// TwinCAT 3 PLC project protobuf
// Title: protobuf
// Company: TcHaxx
// Author: densogiaichned
// ProjectVersion: 0.0.1.0
// Description: Protocol Buffers for TwinCAT 3
// ProgramVersion: 3.1.4026.23
// libraries:
//   snappy, * (TcHaxx)
//   Tc2_Standard, * (Beckhoff Automation GmbH)
//   Tc2_System, * (Beckhoff Automation GmbH)
//   Tc2_Utilities, * (Beckhoff Automation GmbH)
//   TcUnit, * (www.tcunit.org)
// project tree:
//   DUTs/ E_CodedInputStreamErrorCode.TcDUT, E_CodedOutputStreamErrorCode.TcDUT, ST_ParseContext.TcDUT, ST_WriteContext.TcDUT, ST_Span.TcDUT, T_ProtobufMaxString.TcDUT, T_ProtobufRawBuffer.TcDUT
//   FieldCodec/ FB_FieldCodec.TcPOU, FB_FieldCodecFixed32.TcPOU, FB_FieldCodecFixed64.TcPOU, FB_FieldCodecDouble.TcPOU, FB_FieldCodecBool.TcPOU, FB_FieldCodecEnum.TcPOU, FB_FieldCodecMessage.TcPOU, FB_FieldCodecUInt64.TcPOU, FB_FieldCodecUInt32.TcPOU, FB_FieldCodecString.TcPOU, FB_FieldCodecFloat.TcPOU, FB_FieldCodecInt32.TcPOU, FB_FieldCodecSint32.TcPOU, FB_FieldCodecInt64.TcPOU, FB_FieldCodecSint64.TcPOU, FB_FieldCodecBytes.TcPOU
//   GVLs/ GCL_PB.TcGVL, Param_PB.TcGVL
//   Helper/DUTs/ ST_VariableLengthArrayInfo.TcDUT, T_AnyInt.TcDUT, T_AnyIntOrBit.TcDUT, T_AnyString.TcDUT, T_AnyNum.TcDUT, T_Any.TcDUT, T_AnyBit.TcDUT, T_AnyBytes.TcDUT
//   Helper/POUs/ F_ParseError.TcPOU, F_WriteError.TcPOU, F_ToAnyBit.TcPOU, F_ToAnyInt.TcPOU, F_ToAnyBytes.TcPOU, F_ToAnyType.TcPOU, F_ToAnyNum.TcPOU, F_ToAnyString.TcPOU, F_BufferInfo.TcPOU, F_WriteToBuffer.TcPOU, F_ReadFromBuffer.TcPOU
//   ITFs/ I_Message.TcIO, I_FieldCodec.TcIO, I_RepeatedField.TcIO, I_ValueReader.TcIO, I_ValueWriter.TcIO
//   ParsingPrimitivesMessages/POUs/ F_ReadMessage.TcPOU, F_ReadRawMessage.TcPOU, F_SkipLastField.TcPOU, F_CheckReadEndOfStreamTag.TcPOU
//   ParsingPrimitives/DUTs/ E_ParserErrorCode.TcDUT, ST_ParserInternalState.TcDUT
//   ParsingPrimitives/POUs/ F_DecodeZigZag32.TcPOU, F_DecodeZigZag64.TcPOU, F_MaybeConsumeTag.TcPOU, F_ParseDouble.TcPOU, F_ParseFloat.TcPOU, F_ParseRawLittleEndian32.TcPOU, F_ParseLength.TcPOU, F_ParseRawLittleEndian64.TcPOU, F_ParseRawVarint64.TcPOU, F_ParseTag.TcPOU, F_ParseRawVarint32.TcPOU, F_PeekTag.TcPOU, F_ReadBytes.TcPOU, F_ReadRawByte.TcPOU, F_ReadRawBytes.TcPOU, F_ReadStringInternal.TcPOU, F_SkipRawBytes.TcPOU, F_ReadRawString.TcPOU, F_ReadString.TcPOU
//   / PlcTask.TcTTO, PlcTaskUnitTests.TcTTO
//   POUs/ComputeSize/ F_ComputeBoolSize.TcPOU, F_ComputeMessageSize.TcPOU, F_ComputeTagSize.TcPOU, F_ComputeStringSize.TcPOU, F_ComputeFixed32Size.TcPOU, F_ComputeSFixed32Size.TcPOU, F_ComputeFixed64Size.TcPOU, F_ComputeSFixed64Size.TcPOU, F_ComputeInt32Size.TcPOU, F_ComputeEnumSize.TcPOU, F_ComputeFloatSize.TcPOU, F_ComputeDoubleSize.TcPOU, F_ComputeInt64Size.TcPOU, F_ComputeLengthSize.TcPOU, F_ComputeBytesSize.TcPOU, F_ComputeRawVarint64Size.TcPOU, F_ComputeSInt64Size.TcPOU, F_ComputeUInt32Size.TcPOU, F_ComputeRawVarint32Size.TcPOU, F_ComputeSInt32Size.TcPOU, F_ComputeUInt64Size.TcPOU
//   POUs/ FB_MessageParser.TcPOU, FB_MessageWriter.TcPOU
//   POUs/ParseContext/ FB_ParseContext.TcPOU
//   POUs/SegmentedBufferHelper/ F_SbhIsReachedLimit.TcPOU, F_SbhPushLimit.TcPOU, F_SbhPopLimit.TcPOU, F_SbhRecomputeBufferSizeAfterLimit.TcPOU
//   POUs/Span/ F_SpanFromArray.TcPOU, F_SpanSlice.TcPOU
//   POUs/WriteContext/ FB_WriteContext.TcPOU
//   Project Information/ F_GetCompany.TcPOU, F_GetTitle.TcPOU, F_GetVersion.TcPOU
//   RepeatedField/ FB_RepeatedField.TcPOU, F_IsPackedRepeatedField.TcPOU, F_ReadRepeatedField.TcPOU, F_WriteRepeatedField.TcPOU
//   WireFormat/DUTs/ E_WireType.TcDUT
//   WireFormat/GCLs/ GCL_WireFormat.TcGVL
//   WireFormat/POus/ F_GetTagFieldNumber.TcPOU, F_GetTagWireType.TcPOU, F_MakeTag.TcPOU
//   WritingPrimitivesMessages/POUs/ F_SetMessageValue.TcPOU, F_WriteMessage.TcPOU, F_WriteRawMessage.TcPOU
//   WritingPrimitives/DUTs/ E_WriterErrorCode.TcDUT, ST_WriterInternalState.TcDUT
//   WritingPrimitives/POUs/ F_EncodeZigZag32.TcPOU (not stored), F_EncodeZigZag64.TcPOU (not stored), F_WriteBytes.TcPOU, F_WriteDouble.TcPOU, F_WriteFixed32.TcPOU (not stored), F_WriteRawByte.TcPOU, F_WriteSInt32.TcPOU, F_WriteSFixed32.TcPOU (not stored), F_WriteFloat.TcPOU (not stored), F_WriteInt32.TcPOU, F_WriteFixed64.TcPOU (not stored), F_WriteSFixed64.TcPOU (not stored), F_WriteSInt64.TcPOU, F_WriteRawString.TcPOU (not stored), F_WriteRawTag.TcPOU (not stored), F_WriteUInt32.TcPOU (not stored), F_WriteRawLittleEndian32.TcPOU, F_WriteLength.TcPOU, F_WriteRawBytes.TcPOU, F_WriteRawLittleEndian64.TcPOU, F_WriteRawVarint32.TcPOU, F_WriteRawVarint64.TcPOU (not stored), F_WriteString.TcPOU (not stored), F_WriteTag.TcPOU (not stored), F_WriteEnum.TcPOU, F_WriteUInt64.TcPOU (not stored), F_WriteInt64.TcPOU
//   __TESTs/EnumTests/DUTs/ E_INT.TcDUT, E_BYTE.TcDUT
//   __TESTs/EnumTests/ FB_F_ComputeEnumSizeTests.TcPOU, FB_ReadEnumTests.TcPOU, FB_WriteEnumTests.TcPOU, PRG_EnumTests.TcPOU
//   __TESTs/HelperTests/ FB_F_ToAnyBytesTests.TcPOU, PRG_HelperTests.TcPOU
//   __TESTs/MessagesTests/Complex/ FB_ComplexDataTests.TcPOU, FB_RepeatedComplexDataTests.TcPOU, FB_DeviceTests.TcPOU, FB_MotorTests.TcPOU
//   __TESTs/MessagesTests/Complex/_gen/ E_Color.TcDUT, E_DataType.TcDUT, E_Status.TcDUT, FB_ComplexData.TcPOU, FB_Device.TcPOU, FB_Motor.TcPOU, FB_MotorConfig.TcPOU, FB_RepeatedComplexData.TcPOU, FB_SensorReading.TcPOU, ST_ComplexData.TcDUT, ST_Device.TcDUT, ST_Motor.TcDUT, ST_MotorConfig.TcDUT, ST_RepeatedComplexData.TcDUT, ST_SensorReading.TcDUT
//   __TESTs/MessagesTests/DUTs/ ST_Example.TcDUT
//   __TESTs/MessagesTests/FooBarBaz/ FB_FooBarBazTests.TcPOU
//   __TESTs/MessagesTests/FooBarBaz/_gen/ FB_Bar.TcPOU, FB_Baz.TcPOU, FB_Foo.TcPOU, ST_Bar.TcDUT, ST_Baz.TcDUT, ST_Foo.TcDUT
//   __TESTs/MessagesTests/POUs/ FB_ExampleMessage.TcPOU, FB_RoundTripMessageExampleTest.TcPOU
//   __TESTs/MessagesTests/ PRG_MessageTests.TcPOU
//   __TESTs/MessagesTests/Scalars/ FB_ScalarTypesTest.TcPOU
//   __TESTs/MessagesTests/Scalars/_gen/ FB_ScalarTypes.TcPOU, ST_ScalarTypes.TcDUT
//   __TESTs/ParsingPrimitivesTests/ FB_DecodeZigZag32Tests.TcPOU (not stored), FB_DecodeZigZag64Tests.TcPOU (not stored), FB_ParseDoubleTests.TcPOU, FB_ParseFloatTests.TcPOU, FB_ParseRawVarint32Tests.TcPOU, FB_ParseRawVarint64Tests.TcPOU, FB_ReadBytesTests.TcPOU, FB_ReadRawStringTests.TcPOU, FB_ReadStringTests.TcPOU, PRG_ParsingPrimitiveTests.TcPOU
//   __TESTs/ PRG_UnitTests.TcPOU
//   Version/ Global_Version.TcGVL
//   __TESTs/RepeatedFieldTests/ PRG_RepeatedFieldTests.TcPOU
//   __TESTs/RepeatedFieldTests/Read/ FB_ReadRepeatedFieldEnumTests.TcPOU, FB_ReadRepeatedFieldBoolTests.TcPOU, FB_ReadRepeatedFieldBytesTests.TcPOU, FB_ReadRepeatedFieldFixed32Tests.TcPOU, FB_ReadRepeatedFieldFixed64Tests.TcPOU, FB_ReadRepeatedFieldStringTests.TcPOU, FB_ReadRepeatedFieldUint32Tests.TcPOU, PRG_ReadRepeatedFieldTests.TcPOU
//   __TESTs/RepeatedFieldTests/RoundTrip/ FB_RoundTripRepeatedFieldUInt32Tests.TcPOU, FB_RoundTripRepeatedFieldStringTests.TcPOU, FB_RoundTripRepeatedFieldUInt64Tests.TcPOU, PRG_RoundTripRepeatedFieldTests.TcPOU
//   __TESTs/RepeatedFieldTests/Write/ FB_WriteRepeatedFieldBoolTests.TcPOU, FB_WriteRepeatedFieldBytesTests.TcPOU, FB_WriteRepeatedFieldDoubleTests.TcPOU, FB_WriteRepeatedFieldFixed32Tests.TcPOU, FB_WriteRepeatedFieldFixed64Tests.TcPOU, FB_WriteRepeatedFieldFloatTests.TcPOU, FB_WriteRepeatedFieldInt32Tests.TcPOU, FB_WriteRepeatedFieldInt64Tests.TcPOU, FB_WriteRepeatedFieldMessageTests.TcPOU, FB_WriteRepeatedFieldSInt32Tests.TcPOU, FB_WriteRepeatedFieldSInt64Tests.TcPOU, FB_WriteRepeatedFieldStringTests.TcPOU, FB_WriteRepeatedFieldUint32Tests.TcPOU, FB_WriteRepeatedFieldUint64Tests.TcPOU, PRG_WriteRepeatedFieldTests.TcPOU
//   __TESTs/RoundTripTests/ FB_RoundTripBytesTests.TcPOU, FB_RoundTripFloatTests.TcPOU, FB_RoundTripDoubleTests.TcPOU, FB_RoundTripRawVarint32Tests.TcPOU, FB_RoundTripRawVarint64Tests.TcPOU, FB_RoundTripStringTests.TcPOU, FB_RoundTripTagTests.TcPOU, FB_RoundTripZigZag32Tests.TcPOU, FB_RoundTripZigZag64Tests.TcPOU, PRG_RoundTripTests.TcPOU
//   __TESTs/SpanTests/ FB_F_SpanFromArrayTests.TcPOU, FB_F_SpanSliceTests.TcPOU, PRG_SpanTests.TcPOU
//   __TESTs/WireFormatTests/ FB_MakeTagTests.TcPOU, PRG_WireFormatTests.TcPOU
//   __TESTs/WritingPrimitiveTests/ FB_EncodeZigZag64Tests.TcPOU (not stored), FB_EncodeZigZag32Tests.TcPOU, FB_WriteBytesTests.TcPOU, FB_WriteDoubleTests.TcPOU, FB_WriteRawVarint32Tests.TcPOU, FB_WriteFloatTests.TcPOU, FB_WriteRawVarint64Tests.TcPOU, FB_WriteTagTests.TcPOU, FB_WriteStringTests.TcPOU, PRG_WritingPrimitiveTests.TcPOU
//   __TESTs/_ISSUES/ FB_Issue4Tests.TcPOU, PRG_IssuesTests.TcPOU
//   __TESTs/_ISSUES/_gen/ E_EnumOfTypeSint.TcDUT, FB_RepeatedEnumTests.TcPOU, ST_RepeatedEnumTests.TcDUT
// real-time tasks:
//   TASK PlcTask: cycle T#10ms, priority 8, ADS port 350
//   TASK PlcTaskUnitTests: cycle T#10ms, priority 6, ADS port 351

CONFIGURATION protobuf
    RESOURCE PLC ON TwinCAT3
        TASK PlcTask(INTERVAL := T#10ms, PRIORITY := 8);
        TASK PlcTaskUnitTests(INTERVAL := T#10ms, PRIORITY := 6);
        PROGRAM PRG_UnitTests WITH PlcTaskUnitTests : PRG_UnitTests;
    END_RESOURCE
END_CONFIGURATION

// ---- DUTs/E_CodedInputStreamErrorCode.TcDUT
{attribute 'qualified_only'}
{attribute 'strict'}
{attribute 'to_string'}
TYPE E_CodedInputStreamErrorCode :
(
	NoError := S_OK,            // No Error.
    BUFFER_LOWER_BOUND := -1,   // Invalid lower bound for buffer.
    BUFFER_SIZE := -2           // Invalid size of buffer (0 >= size > Param.cMaxProtobufRawBuffer).
) DINT;
END_TYPE

// ---- DUTs/E_CodedOutputStreamErrorCode.TcDUT
{attribute 'qualified_only'}
{attribute 'strict'}
{attribute 'to_string'}
TYPE E_CodedOutputStreamErrorCode :
(
	NoError := S_OK,            // No Error.
    BUFFER_LOWER_BOUND := -1,   // Invalid lower bound for buffer.
    BUFFER_SIZE := -2           // Invalid size of buffer (0 >= size > Param.cMaxProtobufRawBuffer).
) DINT;
END_TYPE

// ---- DUTs/ST_ParseContext.TcDUT
TYPE ST_ParseContext :
STRUCT
    stBuffer    	: ST_Span;
    stState     	: ST_ParserInternalState;
	pCurrentContext : POINTER TO FB_ParseContext; 	// The current context we are operating on
END_STRUCT
END_TYPE

// ---- DUTs/ST_WriteContext.TcDUT
// An opaque struct that represents the current serialization state and is passed along as the serialization proceeds.
TYPE ST_WriteContext :
STRUCT
    stBuffer    	: ST_Span;
    stState     	: ST_WriterInternalState;
	pCurrentContext : POINTER TO FB_WriteContext;	// The current context we are operating on
END_STRUCT
END_TYPE

// ---- DUTs/ST_Span.TcDUT
TYPE ST_Span :
STRUCT
    pBuffer     : POINTER TO BYTE;
    nSize       : UDINT;
END_STRUCT
END_TYPE

// ---- DUTs/T_ProtobufMaxString.TcDUT
TYPE T_ProtobufMaxString : STRING(Param_PB.cMaxCharacter + 1); END_TYPE

// ---- DUTs/T_ProtobufRawBuffer.TcDUT
TYPE T_ProtobufRawBuffer : ARRAY[0..Param_PB.cMaxProtobufRawBuffer] OF BYTE; END_TYPE

// ---- Helper/DUTs/ST_VariableLengthArrayInfo.TcDUT
TYPE ST_VariableLengthArrayInfo :
STRUCT
    nLowerBound : DINT;
    nUpperBound : DINT;
    nSize       : UDINT;
END_STRUCT
END_TYPE

// ---- Helper/DUTs/T_AnyInt.TcDUT
TYPE T_AnyInt : __SYSTEM.AnyType; END_TYPE

// ---- Helper/DUTs/T_AnyIntOrBit.TcDUT
TYPE T_AnyIntOrBit : __SYSTEM.AnyType; END_TYPE

// ---- Helper/DUTs/T_AnyString.TcDUT
TYPE T_AnyString : __SYSTEM.AnyType; END_TYPE

// ---- Helper/DUTs/T_AnyNum.TcDUT
TYPE T_AnyNum : __SYSTEM.AnyType; END_TYPE

// ---- Helper/DUTs/T_Any.TcDUT
TYPE T_Any : __SYSTEM.AnyType; END_TYPE

// ---- Helper/DUTs/T_AnyBit.TcDUT
TYPE T_AnyBit : __SYSTEM.AnyType; END_TYPE

// ---- Helper/DUTs/T_AnyBytes.TcDUT
TYPE T_AnyBytes : __SYSTEM.AnyType; END_TYPE

// ---- ParsingPrimitives/DUTs/E_ParserErrorCode.TcDUT
// Parser ErrorCode is set when a message being parsed is invalid in some way,
// e.g. malformed Varint. Zero means no error.
{attribute 'qualified_only'}
{attribute 'strict'}
{attribute 'to_string'}
TYPE E_ParserErrorCode :
(
	NoError := S_OK,                // No Error.
    InternalError := -1,            // Internal parser error.
    MalformedVarInt := -2,          // Encountered a malformed Varint.
    InvalidDataType := -3,          // Datatype not supported, e.g. F_ParseRawInt32 -> LINT
    TruncatedMessage := -4,         // While parsing a protocol message, the input ended unexpectedly in the middle of a field.  This could mean either that the input has been truncated or that an embedded message misreported its own length.
    InvalidUtf8 := -5,              //
    NotEnoughMem := -6,             // e.g. Array [0..15] OF BYTES but F_ReadRawBytes length is 32.
    EndOfStream := -7,              //
    MoreDataAvailable := -8,        // Completed reading a message while more data was available in the stream.
    RecursionLimitExceeded := -9,   // 
    NegativeSize := -10,            // Encountered an embedded string or message which claimed to have negative size.
    InvalidTag := -11,              // Protocol message contained an invalid tag (zero).
    InvalidWireType := -12,         // Protocol message contained a tag with an invalid wire type.
    NotImplemented := -999          // Not implemented yet.
) DINT := NoError;
END_TYPE

// ---- ParsingPrimitives/DUTs/ST_ParserInternalState.TcDUT
TYPE ST_ParserInternalState :
STRUCT
    nBufferSize             : UDINT;                        // Size of the current buffer
    nBufferPos              : UDINT;                        // The position within the current buffer (i.e. the next byte to read)
    nLastTag                : UDINT;                        // The last tag we read. 0 indicates we've read to the end of the stream (or haven't read anything yet).
    nNextTag                : UDINT;                        //
    nRecursionDepth         : UDINT;                        // Current recursion depth
    nRecursionLimit         : UDINT := Param_PB.cRecursionLimit; 
    nSizeLimit              : UDINT := Param_PB.cMaxProtobufRawBuffer;
    nBufferSizeAfterLimit   : UDINT;                        // If we are currently inside a length-delimited block, this is the number of bytes in the buffer that are still available once we leave the delimited block.
    nCurrentLimit           : UDINT := GCL_PB.cSbhLimit;    // The absolute position of the end of the current length-delimited block (including totalBytesRetired).
    nTotalBytesRetired      : UDINT;                        // The total number of consumed before the start of the current buffer.
    bError                  : BOOL;                         // True if error occured.
    bDiscardUnknownFields   : BOOL;                         // When set to true, unknown fields will be discarded while parsing.
    bHasNextTag             : BOOL; 
    eParserErrorCode        : E_ParserErrorCode;            // 0 = no error, <> 0 = error
END_STRUCT
END_TYPE

// ---- WireFormat/DUTs/E_WireType.TcDUT
// Wire types within protobuf encoding/decoding.
{attribute 'qualified_only'}
{attribute 'to_string'}
TYPE E_WireType :
(
	Varint := 0,            // Variable-length integer.
    Fixed64 := 1,           // Fixed-length 64-bit integer.
    LengthDelimited := 2,   // Length-delimited value, i.e. a length followed by that many bytes of data.
    StartGroup := 3,        // "start group" value
    EndGroup := 4,          // "end group" value
    Fixed32 := 5            // Fixed-length 32-bit value.
) UDINT;
END_TYPE

// ---- WritingPrimitives/DUTs/E_WriterErrorCode.TcDUT
// Wrtier ErrorCode is set when a message being written is invalid in some way,
// e.g. malformed Varint. Zero means no error.
{attribute 'qualified_only'}
{attribute 'strict'}
{attribute 'to_string'}
TYPE E_WriterErrorCode :
(
	NoError := S_OK,            // No Error.
    InternalError := -1,        // Internal writer error.
    MalformedVarInt := -2,      // Encountered a malformed Varint.
    InvalidDataType := -3,      // Datatype not supported, e.g. F_WriteVarInt32 -> LINT
    TruncatedMessage := -4,     // Not enough space left in given buffer
    InvalidUtf8 := -5,          //
    NotEnoughMem := -6          // e.g. Array [0..15] OF BYTES but F_ReadRawBytes length is 32.
) DINT := NoError;
END_TYPE

// ---- WritingPrimitives/DUTs/ST_WriterInternalState.TcDUT
TYPE ST_WriterInternalState :
STRUCT
    nBufferSize         : UDINT;                // Size of the current buffer
    nBufferPos          : UDINT;                // The position within the current buffer (i.e. the next byte to read)
    bError              : BOOL;
    eWriterErrorCode    : E_WriterErrorCode;    // 0 = no error, <> 0 = error
END_STRUCT
END_TYPE

// ---- __TESTs/EnumTests/DUTs/E_INT.TcDUT
{attribute 'qualified_only'}
{attribute 'strict'}
{attribute 'to_string'}
TYPE E_INT :
(	
	eMIN := -32768,
	eVAL0 := 0,
	eVAL1,
	eVAL2,
	eVAL3,
	eMAX := 32767
) INT;
END_TYPE

// ---- __TESTs/EnumTests/DUTs/E_BYTE.TcDUT
{attribute 'qualified_only'}
{attribute 'strict'}
{attribute 'to_string'}
TYPE E_BYTE :
(
	eMIN := 0,
	eVAL1,
	eVAL2,
	eVAL3,
	eMAX := 255
) BYTE;
END_TYPE

// ---- __TESTs/MessagesTests/Complex/_gen/E_Color.TcDUT
(*******************************************************************************
                          protoc-gen-twincat V0.0.0.0                           
                  https://github.com/TcHaxx/protoc-gen-twincat                  
*******************************************************************************)
{attribute 'qualified_only'}
{attribute 'strict'}
{attribute 'to_string'}
// Enum with enum_prefix and enum_integer_type options
TYPE E_Color :
(
	COLOR_DEFAULT := 0,
	COLOR_RED := 1,
	COLOR_GREEN := 2,
	COLOR_BLUE := 3
) WORD;
END_TYPE

// ---- __TESTs/MessagesTests/Complex/_gen/E_DataType.TcDUT
(*******************************************************************************
                          protoc-gen-twincat V0.0.0.0                           
                  https://github.com/TcHaxx/protoc-gen-twincat                  
*******************************************************************************)
{attribute 'qualified_only'}
{attribute 'strict'}
{attribute 'to_string'}
TYPE E_DataType :
(
	DATA_TYPE_UNKNOWN := 0,
	DATA_TYPE_TEMPERATURE := 1,
	DATA_TYPE_PRESSURE := 2,
	DATA_TYPE_HUMIDITY := 3
) BYTE;
END_TYPE

// ---- __TESTs/MessagesTests/Complex/_gen/E_Status.TcDUT
(*******************************************************************************
                          protoc-gen-twincat V0.0.0.0                           
                  https://github.com/TcHaxx/protoc-gen-twincat                  
*******************************************************************************)
{attribute 'qualified_only'}
{attribute 'strict'}
{attribute 'to_string'}
// Another enum for testing
TYPE E_Status :
(
	STATUS_IDLE := 0,
	STATUS_RUNNING := 1,
	STATUS_ERROR := 2
) DWORD;
END_TYPE

// ---- __TESTs/MessagesTests/Complex/_gen/ST_ComplexData.TcDUT
(*******************************************************************************
                          protoc-gen-twincat V0.0.0.0                           
                  https://github.com/TcHaxx/protoc-gen-twincat                  
*******************************************************************************)
{attribute 'no-analysis'}
{attribute 'pack_mode' := '2'}
// Another message demonstrating all field options
TYPE ST_ComplexData :
STRUCT
	label : STRING(512);
	value_dint : DINT;
	value_int : INT;
	value_word : WORD;
	array_data : ARRAY[0..15] OF BYTE;
	array_data_count : UDINT; // Implict generated field for actual number of items in array array_data
	state : E_Status;
	raw_bytes : ARRAY[0..127] OF BYTE;
	raw_bytes_count : UDINT; // Implict generated field for actual number of items in array raw_bytes
	measurement : LREAL;
	calibration_factor : REAL;
	readings : ARRAY[0..31] OF ST_SensorReading;
	readings_count : UDINT; // Implict generated field for actual number of items in array readings
	data_type : E_DataType;
END_STRUCT
END_TYPE

// ---- __TESTs/MessagesTests/Complex/_gen/ST_Device.TcDUT
(*******************************************************************************
                          protoc-gen-twincat V0.0.0.0                           
                  https://github.com/TcHaxx/protoc-gen-twincat                  
*******************************************************************************)
{attribute 'no-analysis'}
{attribute 'pack_mode' := '1'}
// Message with st_prefix and attribute_pack_mode options
TYPE ST_Device :
STRUCT
	name : STRING(256);
	id : DWORD;
	error_codes : ARRAY[0..9] OF WORD;
	error_codes_count : UDINT; // Implict generated field for actual number of items in array error_codes
	temperature : DINT;
	data : ARRAY[0..63] OF BYTE;
	data_count : UDINT; // Implict generated field for actual number of items in array data
END_STRUCT
END_TYPE

// ---- __TESTs/MessagesTests/Complex/_gen/ST_Motor.TcDUT
(*******************************************************************************
                          protoc-gen-twincat V0.0.0.0                           
                  https://github.com/TcHaxx/protoc-gen-twincat                  
*******************************************************************************)
{attribute 'no-analysis'}
{attribute 'pack_mode' := '4'}
// Message with fb_prefix option (function block)
TYPE ST_Motor :
STRUCT
	name : STRING(128);
	status : E_Status;
	speed : DWORD;
	sensor_readings : ARRAY[0..7] OF SINT;
	sensor_readings_count : UDINT; // Implict generated field for actual number of items in array sensor_readings
	config : ARRAY[0..31] OF BYTE;
	config_count : UDINT; // Implict generated field for actual number of items in array config
	motor_config : ST_MotorConfig;
END_STRUCT
END_TYPE

// ---- __TESTs/MessagesTests/Complex/_gen/ST_MotorConfig.TcDUT
(*******************************************************************************
                          protoc-gen-twincat V0.0.0.0                           
                  https://github.com/TcHaxx/protoc-gen-twincat                  
*******************************************************************************)
{attribute 'no-analysis'}
TYPE ST_MotorConfig :
STRUCT
	max_speed : REAL;
	acceleration : LREAL;
	timeout_ms : DWORD;
END_STRUCT
END_TYPE

// ---- __TESTs/MessagesTests/Complex/_gen/ST_RepeatedComplexData.TcDUT
(*******************************************************************************
                          protoc-gen-twincat V0.0.0.0                           
                  https://github.com/TcHaxx/protoc-gen-twincat                  
*******************************************************************************)
{attribute 'no-analysis'}
TYPE ST_RepeatedComplexData :
STRUCT
	complex_data_list : ARRAY[0..4] OF ST_ComplexData;
	complex_data_list_count : UDINT; // Implict generated field for actual number of items in array complex_data_list
END_STRUCT
END_TYPE

// ---- __TESTs/MessagesTests/Complex/_gen/ST_SensorReading.TcDUT
(*******************************************************************************
                          protoc-gen-twincat V0.0.0.0                           
                  https://github.com/TcHaxx/protoc-gen-twincat                  
*******************************************************************************)
{attribute 'no-analysis'}
TYPE ST_SensorReading :
STRUCT
	value : LREAL;
	precision : REAL;
	timestamp : LINT;
END_STRUCT
END_TYPE

// ---- __TESTs/MessagesTests/DUTs/ST_Example.TcDUT
(*******************************************************************************
                          protoc-gen-twincat V0.0.0.0                           
                  https://github.com/TcHaxx/protoc-gen-twincat                  
*******************************************************************************)
{attribute 'no-analysis'}
// This is a message-level comment.
TYPE ST_Example :
STRUCT
	// This is a leading field-level comment,
	// and it continues on the next line.
	sName : STRING(256);	// Trailing comment for field1 (sName).
	aUdintArray : ARRAY[0..6] OF UDINT;	// Trailing comment for field2 (aUdintArray).
	aUdintArray_count	: UDINT;			// Number of items in the array.
	nDInt2 : DINT;	// Trailing comment for field3 (nDInt2).
	sMyString : STRING;
	nFixed64 : ULINT;
	nSFixed64 : LINT;	// Trailing comment for field4 (nSFixed64).
	// Leading comment for field7 (aByteArray),
	// also multiline...
	aByteArray : ARRAY[0..31] OF BYTE;	// Trailing comment for field7 (aByteArray).
	aByteArray_count	: UDINT;			// Number of items in the array.
	fReal : REAL;
	aLReal : ARRAY[0..7] OF LREAL;	// Trailing comment for field9 (fLReal).
	aLReal_count		: UDINT;			// Number of items in the array.
	aBytes : ARRAY[0..15] OF BYTE;	// Fields of type 'bytes' must have a 'array_length' attribute.
	aBytes_count		: UDINT;			// Number of items in the array.
END_STRUCT
END_TYPE

// ---- __TESTs/MessagesTests/FooBarBaz/_gen/ST_Bar.TcDUT
(*******************************************************************************
                          protoc-gen-twincat v0.0.0.0                           
             https://github.bhs-world.com/CorrML/protoc-gen-twincat             
*******************************************************************************)
{attribute 'no-analysis'}
TYPE ST_Bar :
STRUCT
	name : STRING;
	age : UDINT;
	email : STRING;
END_STRUCT
END_TYPE

// ---- __TESTs/MessagesTests/FooBarBaz/_gen/ST_Baz.TcDUT
(*******************************************************************************
                          protoc-gen-twincat v0.0.0.0                           
             https://github.bhs-world.com/CorrML/protoc-gen-twincat             
*******************************************************************************)
{attribute 'no-analysis'}
TYPE ST_Baz :
STRUCT
	value : UDINT;
	name : STRING;
END_STRUCT
END_TYPE

// ---- __TESTs/MessagesTests/FooBarBaz/_gen/ST_Foo.TcDUT
(*******************************************************************************
                          protoc-gen-twincat v0.0.0.0                           
             https://github.bhs-world.com/CorrML/protoc-gen-twincat             
*******************************************************************************)
{attribute 'no-analysis'}
TYPE ST_Foo :
STRUCT
	bar : ST_Bar;
	baz : ARRAY[0..2] OF ST_Baz;
	baz_count : UDINT; // Implict generated field for actual number of items in array baz
END_STRUCT
END_TYPE

// ---- __TESTs/MessagesTests/Scalars/_gen/ST_ScalarTypes.TcDUT
(*******************************************************************************
                          protoc-gen-twincat v0.0.0.0                           
             https://github.bhs-world.com/CorrML/protoc-gen-twincat             
*******************************************************************************)
{attribute 'no-analysis'}
TYPE ST_ScalarTypes :
STRUCT
	double_value : LREAL;
	float_value : REAL;
	int32_value : DINT;
	int32_value_as_word : WORD;
	int64_value : LINT;
	int64_value_as_dint : DINT;
	uint32_value : UDINT;
	uint32_value_as_byte : BYTE;
	uint64_value : ULINT;
	uint64_value_as_dword : DWORD;
	sint32_value : DINT;
	sint64_value : LINT;
	fixed32_value : UDINT;
	fixed64_value : ULINT;
	sfixed32_value : DINT;
	sfixed64_value : LINT;
	bool_value : BOOL;
	string_value : STRING(128);
	bytes_value : ARRAY[0..15] OF BYTE;
	bytes_value_count : UDINT; // Implict generated field for actual number of items in array bytes_value
END_STRUCT
END_TYPE

// ---- __TESTs/_ISSUES/_gen/E_EnumOfTypeSint.TcDUT
(*******************************************************************************
                          protoc-gen-twincat V0.0.0.0                           
                  https://github.com/TcHaxx/protoc-gen-twincat                  
*******************************************************************************)
{attribute 'qualified_only'}
{attribute 'strict'}
{attribute 'to_string'}
TYPE E_EnumOfTypeSint :
(
	VALUE_0 := 0,
	VALUE_1 := 1,
	VALUE_2 := 2,
	VAULE_3 := 3,
	VALUE_MIN := -127,
	VALUE_MAX := 127
) SINT;
END_TYPE

// ---- __TESTs/_ISSUES/_gen/ST_RepeatedEnumTests.TcDUT
(*******************************************************************************
                          protoc-gen-twincat V0.0.0.0                           
                  https://github.com/TcHaxx/protoc-gen-twincat                  
*******************************************************************************)
{attribute 'no-analysis'}
TYPE ST_RepeatedEnumTests :
STRUCT
	enum_values_sint : ARRAY[0..15] OF E_EnumOfTypeSint;
	enum_values_sint_count : UDINT; // Implict generated field for actual number of items in array enum_values_sint
END_STRUCT
END_TYPE

// ---- GVLs/GCL_PB.TcGVL
{attribute 'qualified_only'}
{attribute 'no-analysis'}
VAR_GLOBAL
    cLittleEndian64Size : UDINT := 8;
    cLittleEndian32Size : UDINT := 4;
    cDoubleSize         : UDINT := cLittleEndian64Size;
    cFloatSize          : UDINT := cLittleEndian32Size;
    cBoolSize           : UDINT := 1;
    cSbhLimit           : UDINT := TO_UDINT(-1);
END_VAR

// ---- GVLs/Param_PB.TcGVL
{attribute 'qualified_only'}
VAR_GLOBAL CONSTANT
    cMaxCharacter                   : UDINT(16#FF..16#FFFF) := 16#3FF;          // Default max. character = 1023.
    cMaxProtobufRawBuffer           : UDINT(16#FF..16#FFFF) := 16#1000;         // Default max. raw buffer size = 4096.
    cFieldCodecBytesDefaultSize     : UDINT(16#20..cMaxCharacter) := 16#100;    // Default tmp. buffer size for field codec Bytes.
    cRecursionLimit                 : UDINT(16#1..16#FF) := 16#64;              // Default recursion limit.
END_VAR

// ---- WireFormat/GCLs/GCL_WireFormat.TcGVL
{attribute 'qualified_only'}
VAR_GLOBAL CONSTANT INTERNAL
    cTagTypeBits : UINT := 3;
    cTagTypeMask : UINT := 7;   // (1 << cTagTypeBits) - 1;
END_VAR

// ---- Version/Global_Version.TcGVL
{attribute 'TcGenerated'}
{attribute 'no-analysis'}
{attribute 'linkalways'}
// This function has been automatically generated from the project information.
VAR_GLOBAL CONSTANT
	{attribute 'const_non_replaced'}
	stLibVersion_protobuf : ST_LibVersion := (iMajor := 0, iMinor := 0, iBuild := 1, iRevision := 0, nFlags := 0, sVersion := '0.0.1.0');
END_VAR

// ---- ITFs/I_Message.TcIO
INTERFACE I_Message EXTENDS __System.IQueryInterface

// Calculates the size of this message in Protocol Buffer wire format, in bytes.
METHOD CalculateSize : UDINT
VAR_INPUT
END_VAR
END_METHOD

// Merges the data from the specified coded input stream with the current message.
METHOD MergeFrom : HRESULT
VAR_IN_OUT
    fbParseCtx   : FB_ParseContext;
END_VAR
END_METHOD

PROPERTY INTERNAL MessageValue : T_Any
GET
END_GET
END_PROPERTY

/// Parser for this message.
PROPERTY Parser : REFERENCE TO FB_MessageParser
GET
END_GET
END_PROPERTY

/// Writer for this message.
PROPERTY Writer : REFERENCE TO FB_MessageWriter
GET
END_GET
END_PROPERTY

// Writes the data to the given coded output stream.
METHOD WriteTo : HRESULT
VAR_IN_OUT
    fbWriteCtx	: FB_WriteContext;
END_VAR
END_METHOD

END_INTERFACE

// ---- ITFs/I_FieldCodec.TcIO
INTERFACE I_FieldCodec EXTENDS I_ValueReader, I_ValueWriter

METHOD ABSTRACT CalculatePackedDataSize : HRESULT
VAR_INPUT CONSTANT
    anyFirstElem    : T_Any;
    nLength         : UDINT;    // items to write
END_VAR
VAR_OUTPUT
    nPackedDataSize : UDINT;
END_VAR
END_METHOD

// Gets the end tag of the codec or 0 if there is no end tag
PROPERTY EndTag : UDINT
GET
END_GET
SET
END_SET
END_PROPERTY

PROPERTY ipMessage : I_Message
GET
END_GET
SET
END_SET
END_PROPERTY

METHOD ABSTRACT IsPackedRepeatedField : BOOL
VAR_INPUT
    nTag : UDINT;
END_VAR
END_METHOD

// Gets the tag of the codec.
PROPERTY Tag : UDINT
GET
END_GET
SET
END_SET
END_PROPERTY

END_INTERFACE

// ---- ITFs/I_RepeatedField.TcIO
INTERFACE I_RepeatedField

METHOD CalculatePackedDataSize : HRESULT
VAR_OUTPUT
    nPackedDataSize : UDINT;
END_VAR
END_METHOD

METHOD CalculateSize : HRESULT

VAR_OUTPUT
	nSize : UDINT;
END_VAR
END_METHOD

METHOD ElementAtIndex : T_ANY
VAR_INPUT
	nIndex		: UDINT;
END_VAR
END_METHOD

PROPERTY ipFieldCodec : I_FieldCodec
GET
END_GET
END_PROPERTY

PROPERTY nCapcacity : UDINT
GET
END_GET
END_PROPERTY

PROPERTY nCount : UDINT
GET
END_GET
SET
END_SET
END_PROPERTY

METHOD SetValue : HRESULT
VAR_INPUT
	anyValue	: T_ANY;
END_VAR
END_METHOD

END_INTERFACE

// ---- ITFs/I_ValueReader.TcIO
INTERFACE I_ValueReader

METHOD ABSTRACT ValueReader : HRESULT
VAR_IN_OUT
    stCtx  : ST_ParseContext;
END_VAR
VAR_OUTPUT
    anyOut : T_Any;
END_VAR
END_METHOD

END_INTERFACE

// ---- ITFs/I_ValueWriter.TcIO
INTERFACE I_ValueWriter

METHOD ABSTRACT ValueWriter : HRESULT
VAR_IN_OUT
    stCtx  : ST_WriteContext;
END_VAR
VAR_INPUT
    anyIn : T_ANY;
END_VAR
END_METHOD

END_INTERFACE

// ---- __TESTs/PRG_UnitTests.TcPOU
{attribute 'analysis' := '-33'}
PROGRAM INTERNAL PRG_UnitTests
VAR
{IF defined (UNIT_TEST)}

{END_IF}
END_VAR

{IF defined (UNIT_TEST)}
PRG_ParsingPrimitiveTests();
PRG_RoundTripTests();
PRG_WritingPrimitiveTests();
PRG_MessageTests();
PRG_WireFormatTests();
PRG_EnumTests();
PRG_RepeatedFieldTests();
PRG_HelperTests();
PRG_SpanTests();
PRG_IssuesTests();
TcUnit.RUN();

{END_IF}

END_PROGRAM

// ---- __TESTs/ParsingPrimitivesTests/PRG_ParsingPrimitiveTests.TcPOU
{attribute 'analysis' := '-33'}
PROGRAM INTERNAL PRG_ParsingPrimitiveTests
VAR
{IF defined (UNIT_TEST)}
    fbParseRawInt32Tests        : FB_ParseRawVarint32Tests;
    fbParseRawInt64Tests        : FB_ParseRawVarint64Tests;
    fbWriteRawInt32Tests        : FB_WriteRawVarint32Tests;
    fbWriteRawInt64Tests        : FB_WriteRawVarint64Tests;
    fbReadRawStringStringTests  : FB_ReadRawStringTests;
    fbReadBytesTests            : FB_ReadBytesTests;
    fbReadStringTests           : FB_ReadStringTests;
    fbDecodeZigZag32Tests       : FB_DecodeZigZag32Tests;
    fbDecodeZigZag64Tests       : FB_DecodeZigZag64Tests;
    fbParseFloatTests           : FB_ParseFloatTests;
    fbParseDoubleTests          : FB_ParseDoubleTests;
{END_IF}
END_VAR

END_PROGRAM

// ---- __TESTs/ParsingPrimitivesTests/FB_ParseRawVarint32Tests.TcPOU
FUNCTION_BLOCK INTERNAL FINAL FB_ParseRawVarint32Tests EXTENDS TcUnit.FB_TestSuite


ShouldParseVarintTheory();
ErrorWhenParsingInvalidDataTheory();

METHOD PRIVATE ErrorWhenParsingInvalidData
VAR_IN_OUT CONSTANT
    aBuffer     : ARRAY [*] OF BYTE;    
END_VAR
VAR_INPUT CONSTANT
    nExpectedHR         : HRESULT;
    nBufferPosStart     : UDINT;
    nExpectedBufferPos  : UDINT;
END_VAR
VAR_INST
    fbCtx           : FB_ParseContext;
END_VAR
VAR
    nActualHR       : DINT;
    nActualResult   : UDINT;    
END_VAR
// Arrange
fbCtx.FromBuffer(aBuffer);
fbCtx.refCtx.stState.nBufferPos := nBufferPosStart;

// Act
nActualHR := F_ParseRawVarint32(fbCtx.refCtx, anyVarInt32Result:= nActualResult);

// Assert
AssertEquals_DINT(
    Expected:= nExpectedHR,
    Actual := nActualHR,
    Message:=CONCAT(__POUNAME(), CONCAT(': ', CONCAT('Expected HRESULT ', TO_STRING(nExpectedHR)))));
 
AssertEquals_UDINT(
    Expected:= nExpectedBufferPos,
    Actual:= fbCtx.refCtx.stState.nBufferPos,
    Message:= CONCAT(CONCAT('Expected stState.nBufferPos to equal ', TO_STRING(nExpectedBufferPos)), CONCAT(', for Varint ', TO_STRING(nExpectedHR))));
END_METHOD

METHOD PRIVATE ErrorWhenParsingInvalidDataTheory : REFERENCE TO FB_Test
VAR CONSTANT
    cRawInvalid1       : ARRAY[0..15] OF BYTE := [16#96];
    cRawInvalid2       : ARRAY[0..15] OF BYTE := [16#96, 16#00];
    cRawInvalid3       : ARRAY[0..15] OF BYTE := [16#00, 16#00, 16#00, 16#FF, 16#FF, 16#FF, 16#FF, 16#FF, 16#FF, 16#FF, 16#FF, 16#FF, 16#FF, 16#01];
END_VAR
TEST(__POUNAME());

ErrorWhenParsingInvalidData(aBuffer:= cRawInvalid1, nExpectedHR := E_ParserErrorCode.MalformedVarInt, nBufferPosStart:= 0, nExpectedBufferPos:= 1);
ErrorWhenParsingInvalidData(aBuffer:= cRawInvalid2, nExpectedHR := E_ParserErrorCode.MalformedVarInt, nBufferPosStart:= 0, nExpectedBufferPos:= 1);
ErrorWhenParsingInvalidData(aBuffer:= cRawInvalid3, nExpectedHR := E_ParserErrorCode.MalformedVarInt, nBufferPosStart:= 3, nExpectedBufferPos:= 13);

TEST_FINISHED_NAMED(__POUNAME());
END_METHOD

METHOD PRIVATE ShouldParseVarint
VAR_IN_OUT CONSTANT
    aBuffer     : ARRAY [*] OF BYTE;    
END_VAR
VAR_INPUT CONSTANT
    nExpected           : UDINT;
    nBufferPosStart     : UDINT;
    nExpectedBufferPos  : UDINT;
END_VAR
VAR_INST
    fbCtx           : FB_ParseContext;
END_VAR
VAR
    nActual         : UDINT;  
    hr              : HRESULT;  
END_VAR
// Arrange
fbCtx.FromBuffer(aBuffer);
fbCtx.refCtx.stState.nBufferPos := nBufferPosStart;

// Act
hr := F_ParseRawVarint32(fbCtx.refCtx, anyVarInt32Result:= nActual);

// Assert
AssertEquals_DINT(
    Expected:= S_OK,
    Actual:= hr,
    Message:= 'Expected S_OK instead of error');
    
AssertEquals_UDINT(
    Expected:= nExpected,
    Actual:= nActual,
    Message:= CONCAT('Expected Varint to equal ', TO_STRING(nExpected)));
 
AssertEquals_UDINT(
    Expected:= nExpectedBufferPos,
    Actual:= fbCtx.refCtx.stState.nBufferPos,
    Message:= CONCAT(CONCAT('Expected stState.nBufferPos to equal ', TO_STRING(nExpectedBufferPos)), CONCAT(', for Varint ', TO_STRING(nExpected))));
END_METHOD

METHOD PRIVATE ShouldParseVarintTheory : REFERENCE TO FB_Test
VAR CONSTANT
    cRawValue0          : ARRAY[0..15] OF BYTE := [16#0];
    cRawValue127        : ARRAY[0..15] OF BYTE := [16#00, 16#00, 16#00, 16#7F];
    cRawValue128        : ARRAY[0..15] OF BYTE := [16#80, 16#01];
    cRawValue150        : ARRAY[0..15] OF BYTE := [16#96, 16#01];
    cRawValue65535      : ARRAY[0..15] OF BYTE := [16#FF, 16#FF, 16#03];
    cRawValue502240990  : ARRAY[0..15] OF BYTE := [16#DE, 16#AD, 16#BE, 16#EF, 16#01];
    cRawValueMaxUdint   : ARRAY[0..15] OF BYTE := [16#00, 16#00, 16#00, 16#FF, 16#FF, 16#FF, 16#FF, 16#0F];
    
    // Negative values for int32 field, should have been SInt32 in protofile
    cRawValueNeg1       : ARRAY[0..15] OF BYTE := [16#FF, 16#FF, 16#FF, 16#FF, 16#FF, 16#FF, 16#FF, 16#FF, 16#FF, 16#01];
    cRawValueNeg1337    : ARRAY[0..15] OF BYTE := [16#C7, 16#F5, 16#FF, 16#FF, 16#FF, 16#FF, 16#FF, 16#FF, 16#FF, 16#01];
END_VAR
TEST(__POUNAME());

ShouldParseVarint(aBuffer:= cRawValue0, nExpected:= 0, nBufferPosStart:= 0, nExpectedBufferPos:= 1);
ShouldParseVarint(aBuffer:= cRawValue127, nExpected:= 127, nBufferPosStart:= 3, nExpectedBufferPos:= 4);
ShouldParseVarint(aBuffer:= cRawValue128, nExpected:= 128, nBufferPosStart:= 0, nExpectedBufferPos:= 2);
ShouldParseVarint(aBuffer:= cRawValue150, nExpected:= 150, nBufferPosStart:= 0, nExpectedBufferPos:= 2);
ShouldParseVarint(aBuffer:= cRawValue65535, nExpected:= 65535, nBufferPosStart:= 0, nExpectedBufferPos:= 3);
ShouldParseVarint(aBuffer:= cRawValue502240990, nExpected:= 502240990, nBufferPosStart:= 0, nExpectedBufferPos:= 5);
ShouldParseVarint(aBuffer:= cRawValueMaxUdint, nExpected:= 16#FFFFFFFF, nBufferPosStart:= 3, nExpectedBufferPos:= 8);

ShouldParseVarint(aBuffer:= cRawValueNeg1, nExpected:= TO_UDINT(-1), nBufferPosStart:= 0, nExpectedBufferPos:= 10);
ShouldParseVarint(aBuffer:= cRawValueNeg1337, nExpected:= TO_UDINT(-1337), nBufferPosStart:= 0, nExpectedBufferPos:= 10);
TEST_FINISHED_NAMED(__POUNAME());
END_METHOD

END_FUNCTION_BLOCK

// ---- POUs/ParseContext/FB_ParseContext.TcPOU
// Represents the current parsing state and is passed along
// as the parsing proceeds.
// All the public methods are intended to be invoked only by the generated code,
// users should never invoke them directly.
{attribute 'no_explicit_call' := 'do not call this POU directly'} 
FUNCTION_BLOCK FINAL FB_ParseContext
VAR_INPUT
END_VAR
VAR_OUTPUT
END_VAR
VAR
    stCtx   : ST_ParseContext;
END_VAR

VAR
END_VAR

// Internal-only property; when set to true, unknown fields will be discarded while parsing.
PROPERTY INTERNAL DiscardUnknownFields : BOOL
GET
DiscardUnknownFields := stCtx.stState.bDiscardUnknownFields;
END_GET
SET
stCtx.stState.bDiscardUnknownFields := DiscardUnknownFields;
END_SET
END_PROPERTY

METHOD FromBuffer : HRESULT
VAR_IN_OUT CONSTANT
    aBuffer : ARRAY [*] OF BYTE;
END_VAR

Reset();
Initialize(F_SpanFromArray(aBuffer));
END_METHOD

METHOD INTERNAL Initialize
VAR_INPUT CONSTANT
    stBuffer    : ST_Span;    
END_VAR
stCtx.stBuffer := stBuffer;

stCtx.stState.nBufferSize       := stBuffer.nSize;
stCtx.stState.nSizeLimit        := Param_PB.cMaxProtobufRawBuffer;
stCtx.stState.nRecursionLimit   := Param_PB.cRecursionLimit; 
stCtx.stState.nCurrentLimit     := TO_UDINT(-1);

stCtx.pCurrentContext 			:= THIS;
END_METHOD

// Initialize a ST_ParseContext using existing ST_ParserInternalState,
METHOD INTERNAL InitializeFromState
VAR_IN_OUT CONSTANT
    stState : ST_ParserInternalState;
    stBuffer : ST_Span;    
END_VAR
THIS^.stCtx.stState  := stState;
THIS^.stCtx.stBuffer := stBuffer;

stCtx.pCurrentContext := THIS;
END_METHOD

// Returns the last tag read, OR 0 IF no tags have been read OR we've read beyond the end of the input.
PROPERTY INTERNAL LastTag : UDINT
GET
LastTag := stCtx.stState.nLastTag;
END_GET
END_PROPERTY

METHOD ReadBool : HRESULT
VAR_OUTPUT
    bValue : BOOL;
END_VAR
VAR
    nTmp : BYTE;
END_VAR

ReadBool := F_ParseRawVarint32(THIS^.stCtx, nTmp);
bValue := nTmp <> 0;
END_METHOD

METHOD ReadBytes : HRESULT
VAR_IN_OUT
    aBytes : ARRAY [*] OF BYTE;
END_VAR
VAR_OUTPUT
	nCount : UDINT;
END_VAR

ReadBytes := F_ReadBytes(THIS^.stCtx, aBytes, nLength=> nCount);
END_METHOD

METHOD PUBLIC ReadDouble : HRESULT
VAR_OUTPUT
    fValue : LREAL;
END_VAR

ReadDouble := F_ParseDouble(THIS^.stCtx, fValue=> fValue);
END_METHOD

METHOD PUBLIC ReadEnum : HRESULT
VAR_INPUT
    anyEnum : ANY;
END_VAR
VAR
    nTmp   : DINT;
END_VAR
IF anyEnum.pValue = NULL OR anyEnum.TypeClass <> __SYSTEM.TYPE_CLASS.TYPE_ENUM THEN
	ReadEnum := E_HRESULTAdsErr.INVALIDDATA;
	RETURN;
END_IF

ReadEnum := F_ParseRawVarint32(THIS^.stCtx, nTmp);
MEMSET(destAddr:= anyEnum.pValue, fillByte:= 16#0, n:= TO_UDINT(anyEnum.diSize));
MEMCPY(anyEnum.pValue, srcAddr:= ADR(nTmp), MIN(TO_UDINT(anyEnum.diSize), SIZEOF(nTmp)));
END_METHOD

METHOD PUBLIC ReadFixed32 : HRESULT
VAR_OUTPUT
    nValue : UDINT;
END_VAR

ReadFixed32 := F_ParseRawLittleEndian32(THIS^.stCtx, nValue=> nValue);
END_METHOD

METHOD PUBLIC ReadFixed64 : HRESULT
VAR_OUTPUT
    nValue : ULINT;
END_VAR

ReadFixed64 := F_ParseRawLittleEndian64(THIS^.stCtx, nValue=> nValue);
END_METHOD

METHOD PUBLIC ReadFloat : HRESULT
VAR_OUTPUT
    fValue : REAL;
END_VAR

ReadFloat := F_ParseFloat(THIS^.stCtx, fValue=> fValue);
END_METHOD

METHOD PUBLIC ReadInt32 : HRESULT
VAR_INPUT
    anyDint : ANY;
END_VAR
VAR
    nTmp   : UDINT;
	retVal : UDINT;
END_VAR

ReadInt32 := F_ParseRawVarint32(THIS^.stCtx, nTmp);
retVal := memcpy(destAddr:= anyDint.pValue, srcAddr:= ADR(nTmp), n:= MIN(TO_UDINT(anyDint.diSize), SIZEOF(nTmp)));
IF retVal = 0 THEN
	ReadInt32:= E_HRESULTAdsErr.INVALIDDATA;
END_IF
END_METHOD

METHOD PUBLIC ReadInt64 : HRESULT
VAR_INPUT
    anyLint : ANY;
END_VAR
VAR
    nTmp   : ULINT;
	retVal : UDINT;
END_VAR

ReadInt64 := F_ParseRawVarint64(THIS^.stCtx, nTmp);
retVal := memcpy(destAddr:= anyLint.pValue, srcAddr:= ADR(nTmp), n:= MIN(TO_UDINT(anyLint.diSize), SIZEOF(nTmp)));
IF retVal = 0 THEN
	ReadInt64:= E_HRESULTAdsErr.INVALIDDATA;
END_IF
END_METHOD

// Reads a length for length-delimited data.
METHOD PUBLIC ReadLength : HRESULT
VAR_OUTPUT
    nLength : UDINT;
END_VAR
ReadLength := F_ParseLength(THIS^.stCtx, nLength=> nLength);
END_METHOD

METHOD ReadMessage : HRESULT
VAR_INPUT
    ipMessage : I_Message;
END_VAR

ReadMessage := F_ReadMessage(fbCtx:= THIS^, ipMessage);
END_METHOD

METHOD PUBLIC ReadSFixed32 : HRESULT
VAR_OUTPUT
    nValue : DINT;
END_VAR
VAR
    nTmp : UDINT;
END_VAR

ReadSFixed32 := F_ParseRawLittleEndian32(THIS^.stCtx, nValue=> nTmp);

nValue := TO_DINT(nTmp);
END_METHOD

METHOD PUBLIC ReadSFixed64 : HRESULT
VAR_OUTPUT
    nValue : LINT;
END_VAR
VAR
    nTmp : ULINT;
END_VAR

ReadSFixed64 := F_ParseRawLittleEndian64(THIS^.stCtx, nValue=> nTmp);

nValue := TO_LINT(nTmp);
END_METHOD

METHOD PUBLIC ReadSInt32 : HRESULT
VAR_INPUT
    anyDint : ANY;
END_VAR
VAR
    nTmp   : UDINT;
	nValue : DINT;
	retVal : UDINT;
END_VAR

ReadSInt32 := F_ParseRawVarint32(THIS^.stCtx, nTmp);
nValue := F_DecodeZigZag32(nTmp);
retVal := memcpy(destAddr:= anyDint.pValue, srcAddr:= ADR(nValue), n:= MIN(TO_UDINT(anyDint.diSize), SIZEOF(nValue)));
IF retVal = 0 THEN
	ReadSInt32:= E_HRESULTAdsErr.INVALIDDATA;
END_IF
END_METHOD

METHOD PUBLIC ReadSInt64 : HRESULT
VAR_INPUT
    anyLint : ANY;
END_VAR
VAR
    nTmp   : ULINT;
	nValue : LINT;
	retVal : UDINT;
END_VAR

ReadSInt64 := F_ParseRawVarint64(THIS^.stCtx, nTmp);
nValue := F_DecodeZigZag64(nTmp);
retVal := memcpy(destAddr:= anyLint.pValue, srcAddr:= ADR(nValue), n:= MIN(TO_UDINT(anyLint.diSize), SIZEOF(nValue)));
IF retVal = 0 THEN
	ReadSInt64:= E_HRESULTAdsErr.INVALIDDATA;
END_IF
END_METHOD

METHOD PUBLIC ReadString : HRESULT
VAR_INPUT
    anyStringOut : ANY_STRING;
END_VAR
ReadString := F_ReadString(THIS^.stCtx, F_ToAnyType(anyStringOut));
END_METHOD

// Peeks at the next field tag. this is like calling "ReadTag", but the
// tag is not consumed. (So a subsequent call to "ReadTag" will return the same value.)
METHOD PUBLIC ReadTag : HRESULT
VAR_OUTPUT
    nTag : UDINT;
END_VAR
ReadTag := F_ParseTag(THIS^.stCtx, nTag=>nTag);
END_METHOD

METHOD PUBLIC ReadUint32 : HRESULT
VAR_INPUT
    anyUdint : ANY;
END_VAR
VAR
    nTmp   : UDINT;
	retVal : UDINT;
END_VAR

ReadUint32 := F_ParseRawVarint32(THIS^.stCtx, nTmp);
retVal := memcpy(destAddr:= anyUdint.pValue, srcAddr:= ADR(nTmp), n:= MIN(TO_UDINT(anyUdint.diSize), SIZEOF(nTmp)));
IF retVal = 0 THEN
	ReadUint32:= E_HRESULTAdsErr.INVALIDDATA;
END_IF
END_METHOD

METHOD PUBLIC ReadUint64 : HRESULT
VAR_INPUT
    anyUlint : ANY;
END_VAR
VAR
    nTmp   : ULINT;
	retVal : UDINT;
END_VAR

ReadUint64 := F_ParseRawVarint64(THIS^.stCtx, nTmp);
retVal := memcpy(destAddr:= anyUlint.pValue, srcAddr:= ADR(nTmp), n:= MIN(TO_UDINT(anyUlint.diSize), SIZEOF(nTmp)));
IF retVal = 0 THEN
	ReadUint64:= E_HRESULTAdsErr.INVALIDDATA;
END_IF
END_METHOD

PROPERTY refCtx : REFERENCE TO ST_ParseContext
GET
refCtx REF= THIS^.stCtx ;
END_GET
END_PROPERTY

METHOD PRIVATE Reset
VAR_INPUT
END_VAR

stCtx.stState.bError := FALSE;
stCtx.stState.eParserErrorCode := S_OK;
stCtx.stState.nBufferPos := 0;
stCtx.stState.nBufferSize := 0;
END_METHOD

METHOD SkipLastField : HRESULT
VAR_INPUT
END_VAR

SkipLastField := F_SkipLastField(THIS^.stCtx);
END_METHOD

END_FUNCTION_BLOCK

// ---- POUs/Span/F_SpanFromArray.TcPOU
FUNCTION F_SpanFromArray : ST_Span
VAR_IN_OUT CONSTANT
    aBuffer : ARRAY [*] OF BYTE;
END_VAR
VAR
    stArrayInfo : ST_VariableLengthArrayInfo;
END_VAR


F_SpanFromArray.pBuffer := ADR(aBuffer[LOWER_BOUND(aBuffer, 1)]);
stArrayInfo := F_BufferInfo(aBuffer);
F_SpanFromArray.nSize   := stArrayInfo.nSize;

END_FUNCTION

// ---- Helper/POUs/F_BufferInfo.TcPOU
FUNCTION F_BufferInfo : ST_VariableLengthArrayInfo
VAR_IN_OUT CONSTANT
    aBuffer : ARRAY[*] OF BYTE;
END_VAR
VAR
    pLB : POINTER TO BYTE;
    pUB : POINTER TO BYTE;
    nLB : DINT;
    nUB : DINT;
END_VAR


nLB := LOWER_BOUND(aBuffer, 1);
nUB := UPPER_BOUND(aBuffer, 1);

pLB := ADR(aBuffer[nLB]);
pUB := ADR(aBuffer[nUB]);

F_BufferInfo.nLowerBound    := nLB;
F_BufferInfo.nUpperBound    := nUB;
F_BufferInfo.nSize          := pUB - pLB + 1;

END_FUNCTION

// ---- ParsingPrimitives/POUs/F_ParseRawVarint32.TcPOU
FUNCTION F_ParseRawVarint32 : HRESULT
VAR_IN_OUT      
    stCtx : ST_ParseContext;
END_VAR
VAR_INPUT
    anyVarInt32Result : ANY;
END_VAR
VAR 
    bTmpByte        : BYTE;
    nResult         : UDINT;
    nShift          : UINT := 1;
    i               : UINT;
END_VAR

IF anyVarInt32Result.diSize > SIZEOF(UDINT) THEN
    F_ParseRawVarint32 := F_ParseError(stCtx, E_ParserErrorCode.InvalidDataType);     
    RETURN; 
END_IF


bTmpByte := PBYTE_TO_BYTE(stCtx.stBuffer.pBuffer + stCtx.stState.nBufferPos);

stCtx.stState.nBufferPos := stCtx.stState.nBufferPos + 1;

IF bTmpByte < 16#80 THEN
    nResult := TO_UDINT(bTmpByte);
    MEMMOVE(destAddr:= anyVarInt32Result.pValue, srcAddr:= ADR(nResult), SIZEOF(nResult));
    RETURN;
END_IF 

nResult := bTmpByte AND 16#7F;

{warning 'TODO: MalformedVarInt needs to be compared with C# protobuf}

WHILE (bTmpByte > 16#7F AND stCtx.stState.nBufferPos <= stCtx.stBuffer.nSize AND nShift < 5) DO
    bTmpByte := PBYTE_TO_BYTE(stCtx.stBuffer.pBuffer + stCtx.stState.nBufferPos);
    
    // MalformedVarInt when we encounter zero value, but MSB was set last iteration.
    IF bTmpByte = 0 THEN
        F_ParseRawVarint32 := F_ParseError(stCtx, E_ParserErrorCode.MalformedVarInt);
        nResult := 0;        
        RETURN;
    END_IF
    
    IF nShift = 4 AND bTmpByte >= 16#80 THEN        
        // Likely a negative encoded value, should have been encoded as SInt32 instead (protofile)...
        nResult := nResult OR SHL((bTmpByte AND 16#7F), nShift * 7);
        FOR i:= 0 TO 5 DO
            // Discard upper 32 bits.
            F_ParseRawVarint32 := F_ReadRawByte(stCtx, nByte=> bTmpByte);
            IF bTmpByte < 16#80 THEN                
                JMP _END_FUNCTION;
            END_IF
        END_FOR
        F_ParseRawVarint32 := F_ParseError(stCtx, E_ParserErrorCode.MalformedVarInt);
        nResult := 0;        
        RETURN;
    
    END_IF
        
    nResult := nResult OR SHL((bTmpByte AND 16#7F), nShift * 7); 
    nShift := nShift + 1; 
    stCtx.stState.nBufferPos := stCtx.stState.nBufferPos + 1;
END_WHILE 

_END_FUNCTION:
MEMMOVE(destAddr:= anyVarInt32Result.pValue, srcAddr:= ADR(nResult), SIZEOF(nResult));
F_ParseRawVarint32 := S_OK;

END_FUNCTION

// ---- Helper/POUs/F_ParseError.TcPOU
// Sets the E_ParserErrorCode in the given ST_ParseContext.
FUNCTION F_ParseError : E_ParserErrorCode
VAR_IN_OUT
    stCtx : ST_ParseContext;
END_VAR
VAR_INPUT
    eError : E_ParserErrorCode;
END_VAR


stCtx.stState.bError := TRUE;
stCtx.stState.eParserErrorCode := eError;

F_ParseError := eError;

END_FUNCTION

// ---- ParsingPrimitives/POUs/F_ReadRawByte.TcPOU
FUNCTION INTERNAL F_ReadRawByte : HRESULT
VAR_IN_OUT
    stCtx : ST_ParseContext;
END_VAR
VAR_OUTPUT
    nByte   : BYTE;
END_VAR


IF stCtx.stState.nBufferPos >= stCtx.stState.nBufferSize THEN
    F_ReadRawByte := F_ParseError(stCtx, E_ParserErrorCode.TruncatedMessage);
    RETURN;
END_IF

nByte := PBYTE_TO_BYTE(stCtx.stBuffer.pBuffer + stCtx.stState.nBufferPos);
stCtx.stState.nBufferPos := stCtx.stState.nBufferPos + 1;

END_FUNCTION

// ---- ParsingPrimitives/POUs/F_ReadBytes.TcPOU
// Reads a bytes field value from the input.
FUNCTION F_ReadBytes : HRESULT
VAR_IN_OUT      
    stCtx : ST_ParseContext; 
    aBytes  : ARRAY[*] OF BYTE;
END_VAR
VAR_OUTPUT
	nLength : UDINT;
END_VAR

F_ReadBytes := S_OK;

F_ReadBytes := F_ParseLength(stCtx, nLength=> nLength);
IF FAILED(F_ReadBytes) THEN
    RETURN;
END_IF

F_ReadBytes := F_ReadRawBytes(stCtx, F_ToAnyBytes(aBytes), nLength);

END_FUNCTION

// ---- ParsingPrimitives/POUs/F_ParseLength.TcPOU
// Reads a length for length-delimited data.
FUNCTION F_ParseLength : HRESULT
VAR_IN_OUT      
    stCtx : ST_ParseContext;
END_VAR
VAR_OUTPUT
    nLength : UDINT;
END_VAR


F_ParseLength := F_ParseRawVarint32(stCtx, nLength);

END_FUNCTION

// ---- ParsingPrimitives/POUs/F_ReadRawBytes.TcPOU
// Reads a fixed size of bytes from the input.
FUNCTION F_ReadRawBytes : HRESULT
VAR_IN_OUT      
    stCtx : ST_ParseContext;
END_VAR
VAR_INPUT CONSTANT
    anyBytes : T_AnyBytes;
    nLength : UDINT;
END_VAR

F_ReadRawBytes := S_OK;

IF anyBytes.TypeClass <> __SYSTEM.TYPE_CLASS.TYPE_ARRAY THEN
    F_ReadRawBytes := stCtx.stState.eParserErrorCode := E_ParserErrorCode.InvalidDataType;
    stCtx.stState.bError := TRUE;
    RETURN;  
END_IF

F_ReadRawBytes := F_ReadFromBuffer(stCtx, anyBytes, nLength);

END_FUNCTION

// ---- Helper/POUs/F_ReadFromBuffer.TcPOU
FUNCTION F_ReadFromBuffer : HRESULT
VAR_IN_OUT      
    stCtx : ST_ParseContext;
END_VAR
VAR_INPUT
    anyData       : T_ANY;
    nLength       : UDINT;      // Items to read
END_VAR

IF stCtx.stBuffer.pBuffer = NULL OR stCtx.stBuffer.nSize = 0 THEN
    F_ReadFromBuffer := F_ParseError(stCtx, E_ParserErrorCode.NotEnoughMem);
    RETURN;    
END_IF

IF nLength > stCtx.stState.nBufferSize - stCtx.stState.nBufferPos THEN
    F_ReadFromBuffer := F_ParseError(stCtx, E_ParserErrorCode.TruncatedMessage);
    RETURN;
END_IF

IF nLength > TO_UDINT(anyData.diSize) THEN
    F_ReadFromBuffer := F_ParseError(stCtx, E_ParserErrorCode.NotEnoughMem);
    RETURN;
END_IF

MEMCPY(destAddr:= anyData.pValue, srcAddr:= stCtx.stBuffer.pBuffer + stCtx.stState.nBufferPos, n:= nLength);
stCtx.stState.nBufferPos := stCtx.stState.nBufferPos + nLength;

END_FUNCTION

// ---- Helper/POUs/F_ToAnyBytes.TcPOU
FUNCTION F_ToAnyBytes : T_AnyBytes
VAR_IN_OUT CONSTANT
    aBytes : ARRAY [*] OF BYTE;
END_VAR

VAR 
    pUB : POINTER TO BYTE;
    nLB : DINT;
    nUB : DINT;
END_VAR

F_ToAnyBytes.TypeClass := __SYSTEM.TYPE_CLASS.TYPE_ARRAY;

nLB := LOWER_BOUND(aBytes, 1);
nUB := UPPER_BOUND(aBytes, 1);

F_ToAnyBytes.pValue := ADR(aBytes[nLB]);
pUB := ADR(aBytes[nUB]);

F_ToAnyBytes.diSize := TO_DINT(pUB - F_ToAnyBytes.pValue) + 1;

END_FUNCTION

// ---- ParsingPrimitives/POUs/F_ParseDouble.TcPOU
// Parses a double value.
FUNCTION F_ParseDouble : HRESULT
VAR_IN_OUT      
    stCtx : ST_ParseContext;
END_VAR
VAR_OUTPUT
    fValue : LREAL;
END_VAR
VAR CONSTANT
    cLength : UDINT := SIZEOF(fValue);
END_VAR
VAR
    fTmp : LREAL;
END_VAR


F_ParseDouble := F_ReadFromBuffer(stCtx, F_ToAnyType(fTmp), cLength);

{warning 'TODO: Check for endianess?'}
fValue := fTmp;

END_FUNCTION

// ---- Helper/POUs/F_ToAnyType.TcPOU
FUNCTION F_ToAnyType : T_Any
VAR_INPUT
    anyArg	: ANY;
END_VAR

F_ToAnyType := anyArg;

END_FUNCTION

// ---- ParsingPrimitives/POUs/F_ParseRawLittleEndian32.TcPOU
// Parses a 32-bit little-endian integer.
FUNCTION F_ParseRawLittleEndian32 : HRESULT
VAR_IN_OUT      
    stCtx : ST_ParseContext;
END_VAR
VAR_OUTPUT
    nValue : UDINT;
END_VAR
VAR CONSTANT
    cLength : UDINT := SIZEOF(nValue);
END_VAR


F_ParseRawLittleEndian32 := F_ReadFromBuffer(stCtx, F_ToAnyType(nValue), cLength);

END_FUNCTION

// ---- ParsingPrimitives/POUs/F_ParseRawLittleEndian64.TcPOU
// Parses a 64-bit little-endian integer.
FUNCTION F_ParseRawLittleEndian64 : HRESULT
VAR_IN_OUT      
    stCtx : ST_ParseContext;
END_VAR
VAR_OUTPUT
    nValue : ULINT;
END_VAR
VAR CONSTANT
    cLength : UDINT := SIZEOF(nValue);
END_VAR


F_ParseRawLittleEndian64 :=  F_ReadFromBuffer(stCtx, F_ToAnyType(nValue), cLength);

END_FUNCTION

// ---- ParsingPrimitives/POUs/F_ParseFloat.TcPOU
// Parses a float value.
FUNCTION F_ParseFloat : HRESULT
VAR_IN_OUT      
    stCtx : ST_ParseContext;
END_VAR
VAR_OUTPUT
    fValue : REAL;
END_VAR
VAR CONSTANT
    cLength : UDINT := SIZEOF(fValue);
END_VAR
VAR
    fTmp : REAL;
END_VAR


F_ParseFloat := F_ReadFromBuffer(stCtx, F_ToAnyType(fTmp), cLength);

{warning 'TODO: Check for endianess?'}
fValue := fTmp;

END_FUNCTION

// ---- ParsingPrimitives/POUs/F_ParseRawVarint64.TcPOU
FUNCTION F_ParseRawVarint64 : HRESULT
VAR_IN_OUT      
    stCtx : ST_ParseContext;
END_VAR
VAR_INPUT
    anyVarInt64Result : ANY_INT;
END_VAR
VAR 
    bTmpByte        : BYTE;
    nResult         : ULINT;
    nShift          : UINT := 1;
END_VAR

IF anyVarInt64Result.diSize > SIZEOF(nResult) THEN
    F_ParseRawVarint64 := F_ParseError(stCtx, E_ParserErrorCode.InvalidDataType);   
    RETURN; 
END_IF


bTmpByte := PBYTE_TO_BYTE(stCtx.stBuffer.pBuffer + stCtx.stState.nBufferPos);

stCtx.stState.nBufferPos := stCtx.stState.nBufferPos + 1;

IF bTmpByte < 16#80 THEN
    nResult := TO_UDINT(bTmpByte);
    MEMMOVE(destAddr:= anyVarInt64Result.pValue, srcAddr:= ADR(nResult), SIZEOF(nResult));
    RETURN;
END_IF 

nResult := bTmpByte AND 16#7F;

{warning 'TODO: MalformedVarInt needs to be compared with C# protobuf}

WHILE (bTmpByte > 16#7F AND stCtx.stState.nBufferPos <= stCtx.stBuffer.nSize AND nShift <= 9) DO
    bTmpByte := PBYTE_TO_BYTE(stCtx.stBuffer.pBuffer + stCtx.stState.nBufferPos);
    
    // MalformedVarInt when we reach the theoretical end of Varint64 but still have MSB set.
    IF nShift = 9 AND bTmpByte >= 16#80 THEN
        F_ParseRawVarint64 := F_ParseError(stCtx, E_ParserErrorCode.MalformedVarInt);
        nResult := 0; 
        RETURN;
    END_IF
    
    // MalformedVarInt when we encounter zero value, but MSB was set last iteration.
    IF bTmpByte = 0 THEN
        F_ParseRawVarint64 := F_ParseError(stCtx, E_ParserErrorCode.MalformedVarInt); 
        nResult := 0; 
        RETURN;
    END_IF
    
    nResult := nResult OR SHL(TO_ULINT(bTmpByte AND 16#7F), nShift * 7); 
    nShift := nShift + 1; 
    stCtx.stState.nBufferPos := stCtx.stState.nBufferPos + 1;
END_WHILE 

MEMMOVE(destAddr:= anyVarInt64Result.pValue, srcAddr:= ADR(nResult), SIZEOF(nResult));

F_ParseRawVarint64 := S_OK;

END_FUNCTION

// ---- ParsingPrimitivesMessages/POUs/F_ReadMessage.TcPOU
FUNCTION F_ReadMessage : HRESULT
VAR_IN_OUT
    fbCtx   : FB_ParseContext;     
END_VAR
VAR_INPUT
    iMessage : I_Message;
END_VAR
VAR
    nLength, nOldLength : UDINT;
END_VAR


F_ReadMessage := F_ParseLength(fbCtx.refCtx, nLength=> nLength);
IF FAILED(F_ReadMessage) THEN
    RETURN;
END_IF

IF fbCtx.refCtx.stState.nRecursionDepth >= fbCtx.refCtx.stState.nRecursionLimit THEN
    F_ReadMessage := fbCtx.refCtx.stState.eParserErrorCode := E_ParserErrorCode.RecursionLimitExceeded;
    fbCtx.refCtx.stState.bError := TRUE;
    RETURN;
END_IF


F_ReadMessage := F_SbhPushLimit(fbCtx.refCtx.stState, nLength, nCurrentLimit=> nOldLength);
IF FAILED(F_ReadMessage) THEN
    RETURN;
END_IF

fbCtx.refCtx.stState.nRecursionDepth := fbCtx.refCtx.stState.nRecursionDepth + 1;
F_ReadMessage := F_ReadRawMessage(fbCtx, iMessage);
IF FAILED(F_ReadMessage) THEN
    RETURN;
END_IF

F_ReadMessage := F_CheckReadEndOfStreamTag(fbCtx.refCtx.stState);
IF FAILED(F_ReadMessage) THEN
    RETURN;
END_IF

IF NOT F_SbhIsReachedLimit(fbCtx.refCtx.stState) THEN
    F_ReadMessage := fbCtx.refCtx.stState.eParserErrorCode := E_ParserErrorCode.TruncatedMessage;
    fbCtx.refCtx.stState.bError := TRUE;
    RETURN;
END_IF

fbCtx.refCtx.stState.nRecursionDepth := fbCtx.refCtx.stState.nRecursionDepth - 1;
F_ReadMessage := F_SbhPopLimit(fbCtx.refCtx.stState, nOldLength);

END_FUNCTION

// ---- POUs/SegmentedBufferHelper/F_SbhPushLimit.TcPOU
(*
Sets currentLimit to (current position) + byteLimit. This is called
when descending into a length-delimited embedded message.
The previouslimit is returned.
*)
FUNCTION INTERNAL F_SbhPushLimit : HRESULT
VAR_IN_OUT
    stState     : ST_ParserInternalState;
END_VAR
VAR_INPUT
    nByteLimit  : UDINT;
END_VAR
VAR_OUTPUT
    nCurrentLimit   : UDINT;
END_VAR


nByteLimit := nByteLimit + stState.nTotalBytesRetired + stState.nBufferPos;

nCurrentLimit := stState.nCurrentLimit;

IF nByteLimit > nCurrentLimit THEN
    F_SbhPushLimit := stState.eParserErrorCode := E_ParserErrorCode.TruncatedMessage;
    stState.bError := TRUE;
    RETURN;
END_IF

stState.nCurrentLimit := nByteLimit;
F_SbhPushLimit := F_SbhRecomputeBufferSizeAfterLimit(stState);

stState.nCurrentLimit := nByteLimit;

END_FUNCTION

// ---- POUs/SegmentedBufferHelper/F_SbhRecomputeBufferSizeAfterLimit.TcPOU
FUNCTION INTERNAL F_SbhRecomputeBufferSizeAfterLimit : HRESULT
VAR_IN_OUT
    stState     : ST_ParserInternalState;
END_VAR
VAR
    nBufferEnd  : UDINT;
END_VAR


stState.nBufferSize := stState.nBufferSize + stState.nBufferSizeAfterLimit;

nBufferEnd := stState.nTotalBytesRetired + stState.nBufferSize;

IF nBufferEnd > stState.nCurrentLimit THEN
    stState.nBufferSizeAfterLimit := nBufferEnd - stState.nCurrentLimit;
    stState.nBufferSize := stState.nBufferSize - stState.nBufferSizeAfterLimit;
ELSE
    stState.nBufferSizeAfterLimit := 0;
END_IF

END_FUNCTION

// ---- ParsingPrimitivesMessages/POUs/F_ReadRawMessage.TcPOU
{attribute 'estimated-stack-usage' := '4096'}
FUNCTION F_ReadRawMessage : HRESULT
VAR_IN_OUT
    fbCtx   : FB_ParseContext;     
END_VAR
VAR_INPUT
    iMessage : I_Message;
END_VAR
VAR
    refState : REFERENCE TO ST_ParserInternalState;
END_VAR


refState REF= fbCtx.refCtx.stState;

IF iMessage = 0 THEN
    F_ReadRawMessage := refState.eParserErrorCode := E_ParserErrorCode.InternalError;
    refState.bError := TRUE;
    RETURN;
END_IF

F_ReadRawMessage := iMessage.MergeFrom(fbCtx);

END_FUNCTION

// ---- ParsingPrimitivesMessages/POUs/F_CheckReadEndOfStreamTag.TcPOU
// Verifies that the last call to ReadTag() returned tag 0
FUNCTION INTERNAL F_CheckReadEndOfStreamTag : HRESULT
VAR_IN_OUT
    stState : ST_ParserInternalState;
END_VAR


IF stState.nLastTag <> 0 THEN
    F_CheckReadEndOfStreamTag := stState.eParserErrorCode := E_ParserErrorCode.MoreDataAvailable;
    stState.bError := TRUE;
    RETURN;
END_IF

END_FUNCTION

// ---- POUs/SegmentedBufferHelper/F_SbhIsReachedLimit.TcPOU
// Returns whether or not all the data before the limit has been read.
FUNCTION INTERNAL F_SbhIsReachedLimit : BOOL
VAR_IN_OUT
    stState     : ST_ParserInternalState;
END_VAR
VAR
    nCurrentAbsolutPos : UDINT;
END_VAR


IF stState.nCurrentLimit = GCL_PB.cSbhLimit THEN
    RETURN;
END_IF

nCurrentAbsolutPos := stState.nTotalBytesRetired + stState.nBufferPos;
F_SbhIsReachedLimit := nCurrentAbsolutPos >= stState.nCurrentLimit;

END_FUNCTION

// ---- POUs/SegmentedBufferHelper/F_SbhPopLimit.TcPOU
// Discards the current limit, returning the previous limit.
FUNCTION INTERNAL F_SbhPopLimit : HRESULT
VAR_IN_OUT
    stState     : ST_ParserInternalState;
END_VAR
VAR_INPUT
    nOldLimit   : UDINT;
END_VAR


stState.nCurrentLimit := nOldLimit;
F_SbhPopLimit := F_SbhRecomputeBufferSizeAfterLimit(stState);

END_FUNCTION

// ---- ParsingPrimitives/POUs/F_DecodeZigZag32.TcPOU
// Decode a 32-bit value with ZigZag encoding.
FUNCTION F_DecodeZigZag32 : DINT
VAR_INPUT
    nValue : UDINT;
END_VAR

F_DecodeZigZag32 := TO_DINT(SHR(nValue, UDINT#1) XOR TO_UDINT(-TO_DINT(nValue AND UDINT#1)));

END_FUNCTION

// ---- ParsingPrimitives/POUs/F_DecodeZigZag64.TcPOU
// Decode a 64-bit value with ZigZag encoding.
FUNCTION F_DecodeZigZag64 : LINT
VAR_INPUT
    nValue : ULINT;
END_VAR

F_DecodeZigZag64 := TO_LINT(SHR(nValue, ULINT#1) XOR TO_ULINT(-TO_LINT(nValue AND ULINT#1)));

END_FUNCTION

// ---- ParsingPrimitives/POUs/F_ReadString.TcPOU
// Reads a string field value from the input.
FUNCTION F_ReadString : HRESULT
VAR_IN_OUT      
    stCtx : ST_ParseContext;
END_VAR
VAR_INPUT
    anyStringOut : T_AnyString;
END_VAR
VAR
    nStrLength : UDINT;
END_VAR

F_ReadString := S_OK;

F_ReadString := F_ParseLength(stCtx, nLength=> nStrLength);
IF FAILED(F_ReadString) THEN
    RETURN;
END_IF

F_ReadString := F_ReadRawString(stCtx, nStrLength, anyStringOut);

END_FUNCTION

// ---- ParsingPrimitives/POUs/F_ReadRawString.TcPOU
// Reads a UTF-8 string from the next "length" bytes.
FUNCTION INTERNAL F_ReadRawString : HRESULT
VAR_IN_OUT      
    stCtx : ST_ParseContext;
END_VAR
VAR_INPUT CONSTANT
    nLength : UDINT;       
    stAnyStringOut : T_Any;
END_VAR
VAR
    pNullByte : POINTER TO BYTE;
END_VAR

F_ReadRawString := S_OK;

IF stAnyStringOut.TypeClass = __SYSTEM.TYPE_CLASS.TYPE_WSTRING THEN
    F_ReadRawString := stCtx.stState.eParserErrorCode := E_ParserErrorCode.InvalidDataType;
    stCtx.stState.bError := TRUE;
    RETURN;
END_IF

IF stAnyStringOut.pValue = NULL THEN 
	F_ReadRawString := stCtx.stState.eParserErrorCode := E_ParserErrorCode.InternalError;
    stCtx.stState.bError := TRUE;
    RETURN;
END_IF

IF nLength > TO_UDINT(stAnyStringOut.diSize - 1) OR 
    nLength > stCtx.stState.nBufferSize - stCtx.stState.nBufferPos THEN
    F_ReadRawString := stCtx.stState.eParserErrorCode := E_ParserErrorCode.TruncatedMessage;
    stCtx.stState.bError := TRUE;
    RETURN;  
END_IF

IF nLength = 0 THEN
    pNullByte := stAnyStringOut.pValue;
    pNullByte^ := 16#0;
    RETURN;
END_IF


MEMCPY(destAddr:= stAnyStringOut.pValue, srcAddr:= stCtx.stBuffer.pBuffer + stCtx.stState.nBufferPos, n:=  nLength);
pNullByte := stAnyStringOut.pValue + nLength;
pNullByte^ := 16#0;

stCtx.stState.nBufferPos := stCtx.stState.nBufferPos + nLength;

END_FUNCTION

// ---- ParsingPrimitives/POUs/F_ParseTag.TcPOU
// Parses the next tag.
// If the end of logical stream was reached, an invalid tag of 0 is returned.
FUNCTION F_ParseTag : HRESULT
VAR_IN_OUT
    stCtx : ST_ParseContext;
END_VAR
VAR_OUTPUT
    nTag : UDINT;
END_VAR

VAR
    nTmp : UDINT;
END_VAR


F_ParseTag := S_OK;

// The "nextTag" logic is there only as an optimization for reading non-packed repeated / map
// fields and is strictly speaking not necessary.
IF stCtx.stState.bHasNextTag THEN
    stCtx.stState.nLastTag := stCtx.stState.nNextTag;
    stCtx.stState.bHasNextTag := FALSE;
    nTag := stCtx.stState.nLastTag;
    RETURN;
END_IF

// Optimize for the incredibly common case of having at least two bytes left in the buffer,
// and those two bytes being enough to get the tag. This will be true for fields up to 4095.
IF stCtx.stState.nBufferPos + 2 <= stCtx.stState.nBufferSize THEN
    nTmp := TO_UDINT(PBYTE_TO_BYTE(stCtx.stBuffer.pBuffer + stCtx.stState.nBufferPos));    
    IF nTmp < 16#80 THEN
        stCtx.stState.nLastTag := nTmp;
        stCtx.stState.nBufferPos := stCtx.stState.nBufferPos + 1;
    ELSE
        F_ParseTag := F_ParseRawVarint32(stCtx, nTmp);
        IF FAILED(F_ParseTag) THEN            
            RETURN;
        END_IF
    END_IF
ELSE   
    // is at end?
    IF stCtx.stState.nBufferPos = stCtx.stState.nBufferSize THEN
        nTag := stCtx.stState.nLastTag := 0;
        RETURN;
    END_IF;
    
    F_ParseTag := F_ParseRawVarint32(stCtx, nTmp);
END_IF

nTag := stCtx.stState.nLastTag := nTmp;

END_FUNCTION

// ---- ParsingPrimitivesMessages/POUs/F_SkipLastField.TcPOU
// Reading and skippig messages / groups
FUNCTION INTERNAL F_SkipLastField : HRESULT
VAR_IN_OUT      
    stCtx : ST_ParseContext;
END_VAR
VAR
    nLength : UDINT;
    nDummy  : UDINT;
END_VAR


IF stCtx.stState.nLastTag = 0 THEN
    F_SkipLastField := F_ParseError(stCtx, E_ParserErrorCode.EndOfStream);
    RETURN;
END_IF

CASE F_GetTagWireType(stCtx.stState.nLastTag) OF
    E_WireType.StartGroup,
    E_WireType.EndGroup:
        F_SkipLastField := F_ParseError(stCtx, E_ParserErrorCode.NotImplemented);

    E_WireType.Fixed32:
        F_SkipLastField := F_ParseRawLittleEndian32(stCtx, nValue=> );
       
    E_WireType.Fixed64:
        F_SkipLastField := F_ParseRawLittleEndian64(stCtx, nValue=> );
       
    E_WireType.LengthDelimited:
        F_SkipLastField := F_ParseLength(stCtx, nLength=> nLength);
        IF SUCCEEDED(F_SkipLastField) THEN
            F_SkipLastField := F_SkipRawBytes(nLength, stCtx.stState);
        END_IF
    
    E_WireType.Varint:
        F_SkipLastField := F_ParseRawVarint32(stCtx, nDummy);
ELSE
    F_SkipLastField := F_ParseError(stCtx, E_ParserErrorCode.InternalError);
    RETURN;
END_CASE

END_FUNCTION

// ---- WireFormat/POus/F_GetTagWireType.TcPOU
// Given a tag value, determines the wire type (lower 3 bits).
FUNCTION F_GetTagWireType : E_WireType
VAR_INPUT
    nTag    : UDINT;
END_VAR
VAR
END_VAR

F_GetTagWireType := nTag AND GCL_WireFormat.cTagTypeMask;

END_FUNCTION

// ---- ParsingPrimitives/POUs/F_SkipRawBytes.TcPOU
// Reads and discards fixed size of bytes from the input.
FUNCTION F_SkipRawBytes : HRESULT

VAR_INPUT CONSTANT
    nLength : UDINT;
END_VAR
VAR_IN_OUT
    stState : ST_ParserInternalState;
END_VAR

F_SkipRawBytes := S_OK;

IF nLength > stState.nBufferSize - stState.nBufferPos THEN
    F_SkipRawBytes := stState.eParserErrorCode := E_ParserErrorCode.TruncatedMessage;
    stState.bError := TRUE;
    RETURN;  
END_IF

stState.nBufferPos := stState.nBufferPos + nLength;

END_FUNCTION

// ---- __TESTs/ParsingPrimitivesTests/FB_ParseRawVarint64Tests.TcPOU
FUNCTION_BLOCK INTERNAL FINAL FB_ParseRawVarint64Tests EXTENDS TcUnit.FB_TestSuite


ShouldParseVarintTheory();
ErrorWhenParsingInvalidDataTheory();

METHOD PRIVATE ErrorWhenParsingInvalidData
VAR_IN_OUT CONSTANT
    aBuffer     : ARRAY [*] OF BYTE;    
END_VAR
VAR_INPUT CONSTANT
    nExpectedHR         : HRESULT;
    nBufferPosStart     : UDINT;
    nExpectedBufferPos  : UDINT;
END_VAR
VAR_INST
    fbCtx           : FB_ParseContext;
END_VAR
VAR
    nActualHR       : DINT;
    nActualResult   : ULINT;    
END_VAR
// Arrange
fbCtx.FromBuffer(aBuffer);
fbCtx.refCtx.stState.nBufferPos := nBufferPosStart;

// Act
nActualHR := F_ParseRawVarint64(fbCtx.refCtx, anyVarInt64Result:= nActualResult);

// Assert
AssertEquals_DINT(
    Expected:= nExpectedHR,
    Actual := nActualHR,
    Message:=CONCAT(__POUNAME(), CONCAT(': ', CONCAT('Expected HRESULT ', TO_STRING(nExpectedHR)))));
 
AssertEquals_UDINT(
    Expected:= nExpectedBufferPos,
    Actual:= fbCtx.refCtx.stState.nBufferPos,
    Message:= CONCAT(CONCAT('Expected stState.nBufferPos to equal ', TO_STRING(nExpectedBufferPos)), CONCAT(', for Varint ', TO_STRING(nExpectedHR))));
END_METHOD

METHOD PRIVATE ErrorWhenParsingInvalidDataTheory : REFERENCE TO FB_Test
VAR CONSTANT
    cRawInvalid1       : ARRAY[0..15] OF BYTE := [16#96];
    cRawInvalid2       : ARRAY[0..15] OF BYTE := [16#96, 16#00];
    cRawInvalid3       : ARRAY[0..15] OF BYTE := [16#00, 16#00, 16#00, 16#FF, 16#FF, 16#FF, 16#FF, 16#FF, 16#FF, 16#FF, 16#FF, 16#FF, 16#81];
END_VAR
TEST(__POUNAME());

ErrorWhenParsingInvalidData(aBuffer:= cRawInvalid1, nExpectedHR := E_ParserErrorCode.MalformedVarInt, nBufferPosStart:= 0, nExpectedBufferPos:= 1);
ErrorWhenParsingInvalidData(aBuffer:= cRawInvalid2, nExpectedHR := E_ParserErrorCode.MalformedVarInt, nBufferPosStart:= 0, nExpectedBufferPos:= 1);
ErrorWhenParsingInvalidData(aBuffer:= cRawInvalid3, nExpectedHR := E_ParserErrorCode.MalformedVarInt, nBufferPosStart:= 3, nExpectedBufferPos:= 12);

TEST_FINISHED_NAMED(__POUNAME());
END_METHOD

METHOD PRIVATE ShouldParseVarint
VAR_IN_OUT CONSTANT
    aBuffer     : ARRAY [*] OF BYTE;    
END_VAR
VAR_INPUT CONSTANT
    nExpected           : ULINT;
    nBufferPosStart     : UDINT;
    nExpectedBufferPos  : UDINT;
END_VAR
VAR_INST
    fbCtx           : FB_ParseContext;
END_VAR
VAR    
    nActual         : ULINT;  
    hr              : HRESULT;  
END_VAR
// Arrange
fbCtx.FromBuffer(aBuffer);
fbCtx.refCtx.stState.nBufferPos := nBufferPosStart;

// Act
hr := F_ParseRawVarint64(fbCtx.refCtx, anyVarInt64Result:= nActual);

// Assert
AssertEquals_DINT(
    Expected:= S_OK,
    Actual:= hr,
    Message:= 'Expected S_OK instead of error');
    
AssertEquals_ULINT(
    Expected:= nExpected,
    Actual:= nActual,
    Message:= CONCAT('Expected Varint to equal ', TO_STRING(nExpected)));
 
AssertEquals_UDINT(
    Expected:= nExpectedBufferPos,
    Actual:= fbCtx.refCtx.stState.nBufferPos,
    Message:= CONCAT(CONCAT('Expected stState.nBufferPos to equal ', TO_STRING(nExpectedBufferPos)), CONCAT(', for Varint ', TO_STRING(nExpected))));
END_METHOD

METHOD PRIVATE ShouldParseVarintTheory : REFERENCE TO FB_Test
VAR CONSTANT
    cRawValue0          : ARRAY[0..15] OF BYTE := [16#0];
    cRawValue127        : ARRAY[0..15] OF BYTE := [16#00, 16#00, 16#00, 16#7F];
    cRawValue128        : ARRAY[0..15] OF BYTE := [16#80, 16#01];
    cRawValue150        : ARRAY[0..15] OF BYTE := [16#96, 16#01];
    cRawValue14882      : ARRAY[0..15] OF BYTE := [16#A2, 16#74];
    cRawValue65535      : ARRAY[0..15] OF BYTE := [16#FF, 16#FF, 16#03];
    cRawValue502240990  : ARRAY[0..15] OF BYTE := [16#DE, 16#AD, 16#BE, 16#EF, 16#01];
    cRawValue11964378330978735131 : ARRAY[0..15] OF BYTE := [16#9B, 16#A8, 16#F9, 16#C2, 16#BB, 16#D6, 16#80, 16#85, 16#A6, 16#01];
    cRawValueMaxULint   : ARRAY[0..15] OF BYTE := [16#00, 16#00, 16#00, 16#FF, 16#FF, 16#FF, 16#FF, 16#FF, 16#FF, 16#FF, 16#FF, 16#FF, 16#01];
END_VAR
TEST(__POUNAME());

ShouldParseVarint(aBuffer:= cRawValue0, nExpected:= 0, nBufferPosStart:= 0, nExpectedBufferPos:= 1);
ShouldParseVarint(aBuffer:= cRawValue127, nExpected:= 127, nBufferPosStart:= 3, nExpectedBufferPos:= 4);
ShouldParseVarint(aBuffer:= cRawValue128, nExpected:= 128, nBufferPosStart:= 0, nExpectedBufferPos:= 2);
ShouldParseVarint(aBuffer:= cRawValue150, nExpected:= 150, nBufferPosStart:= 0, nExpectedBufferPos:= 2);
ShouldParseVarint(aBuffer:= cRawValue14882, nExpected:= 14882, nBufferPosStart:= 0, nExpectedBufferPos:= 2);
ShouldParseVarint(aBuffer:= cRawValue65535, nExpected:= 65535, nBufferPosStart:= 0, nExpectedBufferPos:= 3);
ShouldParseVarint(aBuffer:= cRawValue502240990, nExpected:= 502240990, nBufferPosStart:= 0, nExpectedBufferPos:= 5);
ShouldParseVarint(aBuffer:= cRawValue11964378330978735131, nExpected:= 11964378330978735131, nBufferPosStart:= 0, nExpectedBufferPos:= 10);
ShouldParseVarint(aBuffer:= cRawValueMaxULint, nExpected:= 16#FFFFFFFFFFFFFFFF, nBufferPosStart:= 3, nExpectedBufferPos:= 13);

TEST_FINISHED_NAMED(__POUNAME());
END_METHOD

END_FUNCTION_BLOCK

// ---- __TESTs/WritingPrimitiveTests/FB_WriteRawVarint32Tests.TcPOU
FUNCTION_BLOCK INTERNAL FINAL FB_WriteRawVarint32Tests EXTENDS TcUnit.FB_TestSuite
VAR_INPUT
END_VAR
VAR_OUTPUT
END_VAR
VAR
END_VAR

ShouldWriteVarintTheory();

METHOD PRIVATE ShouldWriteVarint
VAR_IN_OUT CONSTANT
    aExpectedBuffer     : ARRAY [*] OF BYTE;    
END_VAR
VAR_INPUT
    nValue              : UDINT;
END_VAR
VAR_INPUT CONSTANT
    nBufferPosStart     : UDINT;
    nExpectedBufferPos  : UDINT;
END_VAR
VAR_INST
    fbCtx   : FB_WriteContext;
END_VAR
VAR
    aActualBuffer       : ARRAY[0..15] OF BYTE; 
    hrActual        : HRESULT;  
END_VAR

// Arrange
fbCtx.FromBuffer(aActualBuffer);
fbCtx.refCtx.stState.nBufferPos := nBufferPosStart;

// Act
hrActual := F_WriteRawVarint32(fbCtx.refCtx, nValue);

// Assert
AssertEquals_DINT(
     Expected:= S_OK,
     Actual:= hrActual,
     Message:= 'Expected S_OK instead of error');

{warning disable C0041}
AssertArrayEquals_BYTE(    
    Expecteds:= aExpectedBuffer,
    Actuals:= aActualBuffer,
    MEssage:= CONCAT('Expected buffers to be equal for Varint ', TO_STRING(nValue))
);

AssertEquals_UDINT(
    Expected:= nExpectedBufferPos,
    Actual:= fbCtx.refCtx.stState.nBufferPos,
    Message:= CONCAT(CONCAT('Expected stState.nBufferPos to equal ', TO_STRING(nExpectedBufferPos)), CONCAT(', for Varint ', TO_STRING(nExpectedBufferPos))));
END_METHOD

METHOD PRIVATE ShouldWriteVarintTheory : REFERENCE TO FB_Test
VAR CONSTANT
    cExpectedRawValue0          : ARRAY[0..15] OF BYTE := [16#0];
    cExpectedRawValue127        : ARRAY[0..15] OF BYTE := [16#00, 16#00, 16#00, 16#7F];
    cExpectedRawValue128        : ARRAY[0..15] OF BYTE := [16#80, 16#01];
    cExpectedRawValue150        : ARRAY[0..15] OF BYTE := [16#96, 16#01];
    cExpectedRawValue65535      : ARRAY[0..15] OF BYTE := [16#FF, 16#FF, 16#03];
    cExpectedRawValue502240990  : ARRAY[0..15] OF BYTE := [16#DE, 16#AD, 16#BE, 16#EF, 16#01];
    cExpectedRawValueMaxUdint   : ARRAY[0..15] OF BYTE := [16#00, 16#00, 16#00, 16#FF, 16#FF, 16#FF, 16#FF, 16#0F];
END_VAR
TEST(__POUNAME());

ShouldWriteVarint(aExpectedBuffer:= cExpectedRawValue0, nValue:= 0, nBufferPosStart:= 0, nExpectedBufferPos:= 1);
ShouldWriteVarint(aExpectedBuffer:= cExpectedRawValue127, nValue:= 127, nBufferPosStart:= 3, nExpectedBufferPos:= 4);
ShouldWriteVarint(aExpectedBuffer:= cExpectedRawValue128, nValue:= 128, nBufferPosStart:= 0, nExpectedBufferPos:= 2);
ShouldWriteVarint(aExpectedBuffer:= cExpectedRawValue150, nValue:= 150, nBufferPosStart:= 0, nExpectedBufferPos:= 2);
ShouldWriteVarint(aExpectedBuffer:= cExpectedRawValue65535, nValue:= 65535, nBufferPosStart:= 0, nExpectedBufferPos:= 3);
ShouldWriteVarint(aExpectedBuffer:= cExpectedRawValue502240990, nValue:= 502240990, nBufferPosStart:= 0, nExpectedBufferPos:= 5);
ShouldWriteVarint(aExpectedBuffer:= cExpectedRawValueMaxUdint, nValue:= 16#FFFFFFFF, nBufferPosStart:= 3, nExpectedBufferPos:= 8);

TEST_FINISHED_NAMED(__POUNAME());
END_METHOD

END_FUNCTION_BLOCK

// ---- POUs/WriteContext/FB_WriteContext.TcPOU
// Represents the current serialization state and is passed along
// as the serialization proceeds.
// All the public methods are intended to be invoked only by the generated code,
// users should never invoke them directly.
{attribute 'no_explicit_call' := 'do not call this POU directly'} 
FUNCTION_BLOCK PUBLIC FINAL FB_WriteContext
VAR
    stCtx   : ST_WriteContext;
END_VAR

VAR
END_VAR

METHOD FromBuffer : HRESULT
VAR_IN_OUT CONSTANT
    aBuffer : ARRAY [*] OF BYTE;
END_VAR

Reset();
Initialize(F_SpanFromArray(aBuffer));
END_METHOD

METHOD INTERNAL Initialize
VAR_INPUT CONSTANT
    stBuffer    : ST_Span;    
END_VAR
stCtx.stBuffer := stBuffer;

stCtx.stState.nBufferSize        := stBuffer.nSize;
stCtx.stState.nBufferPos         := 0;

stCtx.pCurrentContext			:= THIS;
END_METHOD

// Initialize a ST_WriterContext using existing ST_WriterInternalState,
METHOD INTERNAL InitializeFromState
VAR_IN_OUT CONSTANT
    stBuffer : ST_Span;
    stState : ST_WriterInternalState;        
END_VAR
THIS^.stCtx.stState  := stState;
THIS^.stCtx.stBuffer := stBuffer;

stCtx.pCurrentContext := THIS;
END_METHOD

PROPERTY nSpaceLeft : UDINT
GET
nSpaceLeft := stCtx.stState.nBufferSize - stCtx.stState.nBufferPos;
END_GET
END_PROPERTY

PROPERTY refCtx : REFERENCE TO ST_WriteContext
GET
refCtx REF= THIS^.stCtx ;
END_GET
END_PROPERTY

METHOD PRIVATE Reset
VAR_INPUT
END_VAR

stCtx.stState.bError := FALSE;
stCtx.stState.eWriterErrorCode := S_OK;
stCtx.stState.nBufferPos := 0;
stCtx.stState.nBufferSize := 0;
END_METHOD

METHOD WriteBool : HRESULT
VAR_INPUT
    bValue : BOOL;
END_VAR

WriteBool := F_WriteRawByte(THIS^.stCtx, TO_BYTE(bValue));
END_METHOD

METHOD WriteBytes : HRESULT
VAR_IN_OUT CONSTANT
    aBytes  : ARRAY [*] OF BYTE;
END_VAR
VAR_INPUT
    nCount : UDINT;
END_VAR

WriteBytes := F_WriteBytes(THIS^.stCtx, aBytes, nCount);
END_METHOD

METHOD WriteDouble : HRESULT
VAR_INPUT
    fValue : LREAL;
END_VAR
WriteDouble := F_WriteDouble(THIS^.stCtx, fValue);
END_METHOD

METHOD WriteEnum : HRESULT
VAR_INPUT
    anyEnum : ANY;
END_VAR
VAR
	nTmp : DINT;
END_VAR
IF anyEnum.pValue = NULL OR anyEnum.TypeClass <> __SYSTEM.TYPE_CLASS.TYPE_ENUM THEN
	WriteEnum := E_HRESULTAdsErr.INVALIDDATA;
	RETURN;
END_IF

MEMCPY(destAddr:= ADR(nTmp), srcAddr:= anyEnum.pValue, MIN(TO_UDINT(anyEnum.diSize), SIZEOF(nTmp)));
WriteEnum := F_WriteEnum(THIS^.stCtx, nTmp);
END_METHOD

METHOD WriteFixed32 : HRESULT
VAR_INPUT
    nValue : UDINT;
END_VAR

WriteFixed32 := F_WriteFixed32(THIS^.stCtx, nValue);
END_METHOD

METHOD WriteFixed64 : HRESULT
VAR_INPUT
    nValue : ULINT;
END_VAR

WriteFixed64 := F_WriteFixed64(THIS^.stCtx, nValue);
END_METHOD

METHOD WriteFloat : HRESULT
VAR_INPUT
    fValue : REAL;
END_VAR
WriteFloat := F_WriteFloat(THIS^.stCtx, fValue);
END_METHOD

METHOD WriteInt32 : HRESULT
VAR_INPUT
    anyDint : ANY;
END_VAR
VAR
    nTmp   : DINT;
	retVal : UDINT;
END_VAR

retVal := memcpy(destAddr:= ADR(nTmp), srcAddr:= anyDint.pValue, n:= MIN(TO_UDINT(anyDint.diSize), SIZEOF(nTmp)));
IF retVal = 0 THEN
	WriteInt32:= E_HRESULTAdsErr.INVALIDDATA;
	RETURN;
END_IF

WriteInt32 := F_WriteInt32(THIS^.stCtx, nTmp);
END_METHOD

METHOD WriteInt64 : HRESULT
VAR_INPUT
    anyLint : ANY;
END_VAR
VAR
    nTmp   : LINT;
	retVal : UDINT;
END_VAR

retVal := memcpy(destAddr:= ADR(nTmp), srcAddr:= anyLint.pValue, n:= MIN(TO_UDINT(anyLint.diSize), SIZEOF(nTmp)));
IF retVal = 0 THEN
	WriteInt64:= E_HRESULTAdsErr.INVALIDDATA;
	RETURN;
END_IF

WriteInt64 := F_WriteInt64(THIS^.stCtx, nTmp);
END_METHOD

METHOD WriteLength : HRESULT
VAR_INPUT
    nLength : UDINT;
END_VAR

WriteLength := F_WriteLength(THIS^.stCtx, nLength);
END_METHOD

METHOD WriteMessage : HRESULT
VAR_INPUT
    ipMessage : I_Message;
END_VAR

WriteMessage := F_WriteMessage(stCtx:= THIS^.stCtx, ipMessage);
END_METHOD

METHOD WriteRawTag : HRESULT
VAR_INPUT
	nTag    : UDINT;
END_VAR
WriteRawTag := F_WriteRawTag(THIS^.stCtx, nTag);
END_METHOD

METHOD WriteSFixed32 : HRESULT
VAR_INPUT
    nValue : DINT;
END_VAR

WriteSFixed32 := F_WriteSFixed32(THIS^.stCtx, nValue);
END_METHOD

METHOD WriteSFixed64 : HRESULT
VAR_INPUT
    nValue : LINT;
END_VAR

WriteSFixed64 := F_WriteSFixed64(THIS^.stCtx, nValue);
END_METHOD

METHOD WriteSint32 : HRESULT
VAR_INPUT
    anyDint : ANY;
END_VAR
VAR
    nTmp   : DINT;
	retVal : UDINT;
END_VAR

retVal := memcpy(destAddr:= ADR(nTmp), srcAddr:= anyDint.pValue, n:= MIN(TO_UDINT(anyDint.diSize), SIZEOF(nTmp)));
IF retVal = 0 THEN
	WriteSint32:= E_HRESULTAdsErr.INVALIDDATA;
	RETURN;
END_IF

WriteSint32 := F_WriteSInt32(THIS^.stCtx, nTmp);
END_METHOD

METHOD WriteSint64 : HRESULT
VAR_INPUT
    anyLint : ANY;
END_VAR
VAR
    nTmp   : LINT;
	retVal : UDINT;
END_VAR

retVal := memcpy(destAddr:= ADR(nTmp), srcAddr:= anyLint.pValue, n:= MIN(TO_UDINT(anyLint.diSize), SIZEOF(nTmp)));
IF retVal = 0 THEN
	WriteSint64:= E_HRESULTAdsErr.INVALIDDATA;
	RETURN;
END_IF

WriteSint64 := F_WriteSInt64(THIS^.stCtx, nTmp);
END_METHOD

METHOD WriteString : HRESULT
VAR_IN_OUT CONSTANT
    sStringToWrite          : T_ProtobufMaxString;
END_VAR

WriteString := F_WriteString(THIS^.stCtx, sStringToWrite);
END_METHOD

METHOD WriteTag : HRESULT
VAR_INPUT
    nFieldNumber    : UDINT;
    eWireType       : E_WireType;
END_VAR

WriteTag := F_WriteTag(THIS^.stCtx, nFieldNumber, eWireType);
END_METHOD

METHOD WriteUint32 : HRESULT
VAR_INPUT
    anyUdint : ANY;
END_VAR
VAR
    nTmp   : UDINT;
	retVal : UDINT;
END_VAR


retVal := memcpy(destAddr:= ADR(nTmp), srcAddr:= anyUdint.pValue, n:= MIN(TO_UDINT(anyUdint.diSize), SIZEOF(nTmp)));
IF retVal = 0 THEN
	WriteUint32:= E_HRESULTAdsErr.INVALIDDATA;
	RETURN;
END_IF

WriteUint32 := F_WriteUInt32(THIS^.stCtx, nTmp);
END_METHOD

METHOD WriteUint64 : HRESULT
VAR_INPUT
    anyUlint : ANY;
END_VAR
VAR
    nTmp   : ULINT;
	retVal : UDINT;
END_VAR

retVal := memcpy(destAddr:= ADR(nTmp), srcAddr:= anyUlint.pValue, n:= MIN(TO_UDINT(anyUlint.diSize), SIZEOF(nTmp)));
IF retVal = 0 THEN
	WriteUint64:= E_HRESULTAdsErr.INVALIDDATA;
	RETURN;
END_IF

WriteUint64 := F_WriteUInt64(THIS^.stCtx, nTmp);
END_METHOD

END_FUNCTION_BLOCK

// ---- WritingPrimitives/POUs/F_WriteRawByte.TcPOU
// Writes out part of an array of bytes.
FUNCTION F_WriteRawByte : HRESULT
VAR_IN_OUT
    stCtx   : ST_WriteContext;
END_VAR
VAR_INPUT CONSTANT
    nValue  : BYTE;
END_VAR

VAR CONSTANT
    cLength : UDINT := SIZEOF(nValue);
END_VAR
VAR
    pByte   : POINTER TO BYTE;
END_VAR


F_WriteRawByte := S_OK;

IF cLength > stCtx.stState.nBufferSize - stCtx.stState.nBufferPos THEN
    F_WriteRawByte := stCtx.stState.eWriterErrorCode := E_WriterErrorCode.TruncatedMessage;
    stCtx.stState.bError := TRUE;
    RETURN;
END_IF

pByte := stCtx.stBuffer.pBuffer + stCtx.stState.nBufferPos;
pByte^ := nValue;
stCtx.stState.nBufferPos := stCtx.stState.nBufferPos + cLength;

END_FUNCTION

// ---- WritingPrimitives/POUs/F_WriteBytes.TcPOU
// Reads a bytes field value from the input.
FUNCTION F_WriteBytes : HRESULT
VAR_IN_OUT
    stCtx   : ST_WriteContext;
END_VAR
VAR_IN_OUT CONSTANT    
    aBytes  : ARRAY[*] OF BYTE;
END_VAR
VAR_INPUT
    nCount : UDINT;
END_VAR

F_WriteBytes := S_OK;

F_WriteBytes := F_WriteLength(stCtx, nCount);
IF FAILED(F_WriteBytes) THEN
    RETURN;
END_IF

F_WriteBytes := F_WriteRawBytes(stCtx, F_ToAnyBytes(aBytes), nCount);

END_FUNCTION

// ---- WritingPrimitives/POUs/F_WriteLength.TcPOU
// Writes a length (in bytes) for length-delimited data.
FUNCTION F_WriteLength : HRESULT
VAR_IN_OUT
    stCtx   : ST_WriteContext;
END_VAR
VAR_INPUT
    nLength : UDINT;
END_VAR

{warning disable C0041}
F_WriteLength := F_WriteRawVarint32(stCtx, nLength);

END_FUNCTION

// ---- WritingPrimitives/POUs/F_WriteRawVarint32.TcPOU
FUNCTION F_WriteRawVarint32 : HRESULT
VAR_IN_OUT      
    stCtx : ST_WriteContext;
END_VAR
VAR_INPUT
    anyVarInt32 : ANY_INT;
END_VAR
VAR
    nValue  : UDINT;
    pByte   : POINTER TO BYTE;
END_VAR


IF anyVarInt32.diSize > SIZEOF(UDINT) THEN
    F_WriteRawVarint32 := stCtx.stState.eWriterErrorCode := E_WriterErrorCode.InvalidDataType;     
    stCtx.stState.bError := TRUE;
    RETURN; 
END_IF

// Enough capacity left for theoretical max Varint32?
IF (stCtx.stState.nBufferPos + SIZEOF(nValue) + 1) > stCtx.stState.nBufferSize THEN
    F_WriteRawVarint32 := stCtx.stState.eWriterErrorCode := E_WriterErrorCode.TruncatedMessage;     
    stCtx.stState.bError := TRUE;
    RETURN; 
END_IF

nValue := PUDINT_TO_UDINT(in:= anyVarInt32.pValue);

pByte := stCtx.stBuffer.pBuffer + stCtx.stState.nBufferPos;

// fastpath for a common case of single byte value
IF nValue < 16#80 THEN
    pByte^ :=  TO_BYTE(nValue);
    stCtx.stState.nBufferPos := stCtx.stState.nBufferPos + 1;
    F_WriteRawVarint32 := S_OK;
    RETURN;
END_IF

WHILE (stCtx.stState.nBufferPos < stCtx.stState.nBufferSize) DO
    pByte := stCtx.stBuffer.pBuffer + stCtx.stState.nBufferPos;
    IF nValue > 16#7F THEN
        pByte^ := TO_BYTE((nValue AND 16#7F) OR 16#80);
        nValue := SHR(nValue, 7);
        stCtx.stState.nBufferPos := stCtx.stState.nBufferPos + 1;
    ELSE
        pByte^ := TO_BYTE(nValue);
        stCtx.stState.nBufferPos := stCtx.stState.nBufferPos + 1;
        F_WriteRawVarint32 := S_OK;
        RETURN;
    END_IF
END_WHILE

// should never reach
F_WriteRawVarint32 := E_WriterErrorCode.InternalError;

END_FUNCTION

// ---- WritingPrimitives/POUs/F_WriteRawBytes.TcPOU
// Writes out part of an array of bytes.
FUNCTION F_WriteRawBytes : HRESULT
VAR_IN_OUT      
    stCtx : ST_WriteContext;
END_VAR
VAR_INPUT CONSTANT
    tBytes  : T_AnyBytes;
    nLength : UDINT;
END_VAR


F_WriteRawBytes := S_OK;

F_WriteRawBytes := F_WriteToBuffer(stCtx, tBytes, nLength);

END_FUNCTION

// ---- Helper/POUs/F_WriteToBuffer.TcPOU
FUNCTION F_WriteToBuffer : HRESULT
VAR_IN_OUT      
    stCtx : ST_WriteContext;
END_VAR
VAR_INPUT
    anyData       : T_ANY;
    nLength       : UDINT;      // Items to write 
END_VAR

IF stCtx.stBuffer.pBuffer = NULL OR stCtx.stBuffer.nSize = 0 THEN
    F_WriteToBuffer := stCtx.stState.eWriterErrorCode := E_WriterErrorCode.NotEnoughMem;
    stCtx.stState.bError := TRUE;
    RETURN;    
END_IF

IF nLength > stCtx.stState.nBufferSize - stCtx.stState.nBufferPos THEN
    F_WriteToBuffer := stCtx.stState.eWriterErrorCode := E_WriterErrorCode.TruncatedMessage;
    stCtx.stState.bError := TRUE;
    RETURN;
END_IF

IF nLength > TO_UDINT(anyData.diSize) THEN
    F_WriteToBuffer := stCtx.stState.eWriterErrorCode := E_WriterErrorCode.NotEnoughMem;
    stCtx.stState.bError := TRUE;
    RETURN;
END_IF

MEMCPY(destAddr:= stCtx.stBuffer.pBuffer + stCtx.stState.nBufferPos, srcAddr:= anyData.pValue, n:=  nLength);
stCtx.stState.nBufferPos := stCtx.stState.nBufferPos + nLength;

END_FUNCTION

// ---- WritingPrimitives/POUs/F_WriteDouble.TcPOU
// Writes a double field value, without a tag, to the stream.
FUNCTION F_WriteDouble : HRESULT
VAR_IN_OUT
    stCtx   : ST_WriteContext;
END_VAR
VAR_INPUT CONSTANT
    fValue : LREAL;
END_VAR
VAR CONSTANT
    cLength : UDINT := SIZEOF(fValue);
END_VAR
VAR
    fTmp : LREAL;
END_VAR

{warning 'TODO: Check for endianess?'}
fTmp := fValue;

F_WriteDouble := F_WriteToBuffer(stCtx, F_ToAnyType(fTmp), cLength);

END_FUNCTION

// ---- WritingPrimitives/POUs/F_WriteEnum.TcPOU
// Writes an enum value, without a tag, to the stream.
FUNCTION F_WriteEnum : HRESULT
VAR_IN_OUT      
    stCtx : ST_WriteContext;
END_VAR
VAR_INPUT
    nValue : DINT;
END_VAR
VAR
END_VAR


F_WriteEnum := F_WriteInt32(stCtx, nValue);

END_FUNCTION

// ---- WritingPrimitives/POUs/F_WriteInt32.TcPOU
// Writes an int32 field value, without a tag, to the stream.
FUNCTION F_WriteInt32 : HRESULT
VAR_IN_OUT
    stCtx   : ST_WriteContext;
END_VAR
VAR_INPUT
    nValue : DINT;
END_VAR
VAR
    nValueTmp : ULINT;
END_VAR

IF nValue >= 0 THEN
    F_WriteInt32 := F_WriteRawVarint32(stCtx, nValue);
ELSE
    // Must sign-extend.
    nValueTmp := TO_ULINT(nValue);
    F_WriteInt32 := F_WriteRawVarint64(stCtx, nValueTmp);
END_IF

END_FUNCTION

// ---- WritingPrimitives/POUs/F_WriteInt64.TcPOU
// Writes an int64 field value, without a tag, to the stream.
FUNCTION F_WriteInt64 : HRESULT
VAR_IN_OUT
    stCtx   : ST_WriteContext;
END_VAR
VAR_INPUT
    nValue : LINT;
END_VAR
VAR
END_VAR

F_WriteInt64 := F_WriteRawVarint64(stCtx, nValue);

END_FUNCTION

// ---- WritingPrimitivesMessages/POUs/F_WriteMessage.TcPOU
// Writes a message, without a tag. The data is length-prefixed.
FUNCTION F_WriteMessage : HRESULT
VAR_IN_OUT
//     fbCtx   : FB_WriteContext;
	stCtx : ST_WriteContext;     
END_VAR
VAR_INPUT
    ipMessage : I_Message;
END_VAR
VAR
	nLength : UDINT;
END_VAR

IF ipMessage = NULL THEN
	F_WriteMessage := F_WriteError(stCtx:= stCtx, eError:= E_WriterErrorCode.InternalError);
	RETURN;
END_IF

nLength := ipMessage.CalculateSize();
F_WriteMessage := F_WriteLength(stCtx:= stCtx, nLength);
IF FAILED(F_WriteMessage) THEN
	RETURN;
END_IF

F_WriteMessage := F_WriteRawMessage(stCtx, ipMessage);

END_FUNCTION

// ---- Helper/POUs/F_WriteError.TcPOU
// Sets the E_WriterErrorCode in the given ST_WriteContext.
FUNCTION F_WriteError : E_WriterErrorCode
VAR_IN_OUT
    stCtx : ST_WriteContext;
END_VAR
VAR_INPUT
    eError : E_WriterErrorCode;
END_VAR


stCtx.stState.bError := TRUE;
stCtx.stState.eWriterErrorCode := eError;

F_WriteError := eError;

END_FUNCTION

// ---- WritingPrimitivesMessages/POUs/F_WriteRawMessage.TcPOU
// Writes a message, without a tag. Message will be written without a length prefix.
FUNCTION F_WriteRawMessage : HRESULT
VAR_IN_OUT
    stCtx	: ST_WriteContext;    
END_VAR
VAR_INPUT
    ipMessage : I_Message;
END_VAR

IF ipMessage = NULL OR stCtx.pCurrentContext = NULL THEN
	F_WriteRawMessage := F_WriteError(stCtx:= stCtx, eError:= E_WriterErrorCode.InternalError);
	RETURN;
END_IF

F_WriteRawMessage := ipMessage.WriteTo(fbWriteCtx:= stCtx.pCurrentContext^);

END_FUNCTION

// ---- WritingPrimitives/POUs/F_WriteSInt32.TcPOU
// Writes an sint32 value, without a tag, to the stream.
FUNCTION F_WriteSInt32 : HRESULT
VAR_IN_OUT      
    stCtx : ST_WriteContext;
END_VAR
VAR_INPUT
    nValue : DINT;
END_VAR
VAR
    nTmp : UDINT;
END_VAR

nTmp := F_EncodeZigZag32(nValue);
F_WriteSInt32 := F_WriteRawVarint32(stCtx, nTmp);

END_FUNCTION

// ---- WritingPrimitives/POUs/F_WriteSInt64.TcPOU
// Writes an sint64 value, without a tag, to the stream.
FUNCTION F_WriteSInt64 : HRESULT
VAR_IN_OUT      
    stCtx : ST_WriteContext;
END_VAR
VAR_INPUT
    nValue : LINT;
END_VAR
VAR
    nTMP : ULINT;
END_VAR

nTmp := F_EncodeZigZag64(nValue);
F_WriteSInt64 := F_WriteRawVarint64(stCtx, nTmp);

END_FUNCTION

// ---- __TESTs/WritingPrimitiveTests/FB_WriteRawVarint64Tests.TcPOU
FUNCTION_BLOCK INTERNAL FINAL FB_WriteRawVarint64Tests EXTENDS TcUnit.FB_TestSuite
VAR_INPUT
END_VAR
VAR_OUTPUT
END_VAR
VAR
END_VAR

ShouldWriteVarintTheory();

METHOD PRIVATE ShouldWriteVarint
VAR_IN_OUT CONSTANT
    aExpectedBuffer     : ARRAY [*] OF BYTE;    
END_VAR
VAR_INPUT
    nValue              : ULINT;
END_VAR
VAR_INPUT CONSTANT
    nBufferPosStart     : UDINT;
    nExpectedBufferPos  : UDINT;
END_VAR
VAR_INST
    fbCtx   : FB_WriteContext;
END_VAR
VAR
    aActualBuffer       : ARRAY[0..15] OF BYTE; 
    hrActual        : HRESULT;  
END_VAR

// Arrange
fbCtx.FromBuffer(aActualBuffer);
fbCtx.refCtx.stState.nBufferPos := nBufferPosStart;

// Act
hrActual := F_WriteRawVarint64(fbCtx.refCtx, nValue);

// Assert
AssertEquals_DINT(
     Expected:= S_OK,
     Actual:= hrActual,
     Message:= 'Expected S_OK instead of error');

{warning disable C0041}
AssertArrayEquals_BYTE(    
    Expecteds:= aExpectedBuffer,
    Actuals:= aActualBuffer,
    MEssage:= CONCAT('Expected buffers to be equal for Varint ', TO_STRING(nValue))
);

AssertEquals_UDINT(
    Expected:= nExpectedBufferPos,
    Actual:= fbCtx.refCtx.stState.nBufferPos,
    Message:= CONCAT(CONCAT('Expected stState.nBufferPos to equal ', TO_STRING(nExpectedBufferPos)), CONCAT(', for Varint ', TO_STRING(nExpectedBufferPos))));
END_METHOD

METHOD PRIVATE ShouldWriteVarintTheory : REFERENCE TO FB_Test
VAR CONSTANT
    cExpectedRawValue0          : ARRAY[0..15] OF BYTE := [16#0];
    cExpectedRawValue127        : ARRAY[0..15] OF BYTE := [16#00, 16#00, 16#00, 16#7F];
    cExpectedRawValue128        : ARRAY[0..15] OF BYTE := [16#80, 16#01];
    cExpectedRawValue150        : ARRAY[0..15] OF BYTE := [16#96, 16#01];
    cExpectedRawValue14882      : ARRAY[0..15] OF BYTE := [16#A2, 16#74];
    cExpectedRawValue65535      : ARRAY[0..15] OF BYTE := [16#FF, 16#FF, 16#03];
    cExpectedRawValue502240990  : ARRAY[0..15] OF BYTE := [16#DE, 16#AD, 16#BE, 16#EF, 16#01];
    cExpectedRawValue11964378330978735131 : ARRAY[0..15] OF BYTE := [16#9B, 16#A8, 16#F9, 16#C2, 16#BB, 16#D6, 16#80, 16#85, 16#A6, 16#01];
    cExpectedRawValueMaxUdint   : ARRAY[0..15] OF BYTE := [16#00, 16#00, 16#00, 16#FF, 16#FF, 16#FF, 16#FF, 16#FF, 16#FF, 16#FF, 16#FF, 16#FF, 16#01];
END_VAR
TEST(__POUNAME());

ShouldWriteVarint(aExpectedBuffer:= cExpectedRawValue0, nValue:= 0, nBufferPosStart:= 0, nExpectedBufferPos:= 1);
ShouldWriteVarint(aExpectedBuffer:= cExpectedRawValue127, nValue:= 127, nBufferPosStart:= 3, nExpectedBufferPos:= 4);
ShouldWriteVarint(aExpectedBuffer:= cExpectedRawValue128, nValue:= 128, nBufferPosStart:= 0, nExpectedBufferPos:= 2);
ShouldWriteVarint(aExpectedBuffer:= cExpectedRawValue150, nValue:= 150, nBufferPosStart:= 0, nExpectedBufferPos:= 2);
ShouldWriteVarint(aExpectedBuffer:= cExpectedRawValue14882, nValue:= 14882, nBufferPosStart:= 0, nExpectedBufferPos:= 2);
ShouldWriteVarint(aExpectedBuffer:= cExpectedRawValue65535, nValue:= 65535, nBufferPosStart:= 0, nExpectedBufferPos:= 3);
ShouldWriteVarint(aExpectedBuffer:= cExpectedRawValue502240990, nValue:= 502240990, nBufferPosStart:= 0, nExpectedBufferPos:= 5);
ShouldWriteVarint(aExpectedBuffer:= cExpectedRawValue11964378330978735131, nValue:= 11964378330978735131, nBufferPosStart:= 0, nExpectedBufferPos:= 10);
ShouldWriteVarint(aExpectedBuffer:= cExpectedRawValueMaxUdint, nValue:= 16#FFFFFFFFFFFFFFFF, nBufferPosStart:= 3, nExpectedBufferPos:= 13);

TEST_FINISHED_NAMED(__POUNAME());
END_METHOD

END_FUNCTION_BLOCK

// ---- __TESTs/ParsingPrimitivesTests/FB_ReadRawStringTests.TcPOU
FUNCTION_BLOCK INTERNAL FINAL FB_ReadRawStringTests EXTENDS FB_TestSuite
VAR_INPUT
END_VAR
VAR_OUTPUT
END_VAR
VAR
END_VAR

ShouldReadRawStringTheory();

METHOD PRIVATE ShouldReadRawString
VAR_IN_OUT CONSTANT
    aBuffer         : ARRAY[*] OF BYTE;
    sExpectedString : T_MAXSTRING;
END_VAR
VAR_INPUT CONSTANT
    nBufferPosStart     : UDINT;
    nExpectedBufferPos  : UDINT;
END_VAR
VAR_INST
    fbCtx           : FB_ParseContext;
END_VAR
VAR    
    hrActual : HRESULT; 
    // '--- ' to check for null-byte!
    sActual : T_MAXSTRING := '--------------------------------------------------------------------------------------------------------------------------------------------------------------------------------------------------------------------------------------------------------------';
END_VAR

// Arrange
fbCtx.FromBuffer(aBuffer);
fbCtx.refCtx.stState.nBufferPos := nBufferPosStart;

// Act
{warning disable C0041}
hrActual := F_ReadRawString(stCtx:=fbCtx.refCtx, LEN2(ADR(sExpectedString)), F_ToAnyType(sActual));

// Assert
AssertEquals_DINT(
     Expected:= S_OK,
     Actual:= hrActual,
     Message:= 'Expected S_OK instead of error');
AssertEquals_STRING(
    Expected:= sExpectedString,
    Actual:= sActual,
    Message:= '');
AssertEquals_UDINT(
    Expected:= nExpectedBufferPos,
    Actual:= fbCtx.refCtx.stState.nBufferPos,
    Message:= CONCAT(CONCAT('Expected stState.nBufferPos to equal ', TO_STRING(nExpectedBufferPos)), CONCAT(', for String ', LEFT(sExpectedString, 32))));
END_METHOD

METHOD PRIVATE ShouldReadRawStringTheory
VAR CONSTANT
    cRawString_Empty    : ARRAY[0..255] OF BYTE := [16#0];
    cRawString_Space    : ARRAY[0..255] OF BYTE := [16#20];
    cRawString_012345   : ARRAY[0..255] OF BYTE := [16#00, 16#00, 16#30, 16#31, 16#32, 16#33, 16#34, 16#35];
    cRawString_UTF8     : ARRAY[0..255] OF BYTE := [16#75, 16#74, 16#66, 16#2D, 16#38, 16#3A, 16#20, 16#61, 16#2D, 16#7A, 16#2C, 16#20, 16#41, 16#2D, 16#5A, 16#2C, 16#20, 16#30, 16#2D, 16#39, 16#2C, 16#20, 16#C3, 16#A4, 16#C3, 16#84, 16#C3, 16#B6, 16#C3, 16#96, 16#C3, 16#BC, 16#C3, 16#9C, 16#C3, 16#9F, 16#F0, 16#9F, 16#9A, 16#80];
END_VAR
TEST(__POUNAME());

ShouldReadRawString(aBuffer:= cRawString_Empty, sExpectedString:= '', nBufferPosStart:= 0, nExpectedBufferPos:= 0); 
ShouldReadRawString(aBuffer:= cRawString_Space, sExpectedString:= ' ', nBufferPosStart:= 0, nExpectedBufferPos:= 1); 
ShouldReadRawString(aBuffer:= cRawString_012345, sExpectedString:= '012345', nBufferPosStart:= 2, nExpectedBufferPos:= 8); 
ShouldReadRawString(aBuffer:= cRawString_UTF8, sExpectedString:= 'utf-8: a-z, A-Z, 0-9, äÄöÖüÜß🚀', nBufferPosStart:= 0, nExpectedBufferPos:= 40);
 
TEST_FINISHED_NAMED(__POUNAME());
END_METHOD

END_FUNCTION_BLOCK

// ---- __TESTs/ParsingPrimitivesTests/FB_ReadBytesTests.TcPOU
FUNCTION_BLOCK INTERNAL FINAL FB_ReadBytesTests EXTENDS FB_TestSuite
VAR_INPUT
END_VAR
VAR_OUTPUT
END_VAR
VAR
END_VAR

ShouldReadBytesTheory();

METHOD PRIVATE ShouldReadBytes
VAR_IN_OUT CONSTANT
    aBuffer         : ARRAY[*] OF BYTE;
    aExpectedBytes  : ARRAY[0..31] OF BYTE;
END_VAR
VAR_INPUT CONSTANT
    nBufferPosStart     : UDINT;
    nExpectedBufferPos  : UDINT;
END_VAR
VAR_INST
    fbCtx           : FB_ParseContext;
END_VAR
VAR
    aActualBytes : ARRAY[0..31] OF BYTE;
    hrActual : HRESULT; 
END_VAR

// Arrange
fbCtx.FromBuffer(aBuffer);
fbCtx.refCtx.stState.nBufferPos := nBufferPosStart;


// Act
{warning disable C0041}
hrActual := F_ReadBytes(fbCtx.refCtx, aActualBytes);

// Assert
AssertEquals_DINT(
     Expected:= S_OK,
     Actual:= hrActual,
     Message:= 'Expected S_OK instead of error');

AssertArrayEquals_BYTE(
    Expecteds:= aExpectedBytes,
    Actuals:= aActualBytes,
    Message:= '');
    
AssertEquals_UDINT(
    Expected:= nExpectedBufferPos,
    Actual:= fbCtx.refCtx.stState.nBufferPos,
    Message:= CONCAT('Expected stState.nBufferPos to equal ', TO_STRING(nExpectedBufferPos)));
END_METHOD

METHOD PRIVATE ShouldReadBytesTheory
VAR CONSTANT
    cRawBytesTest1          : ARRAY [0..31] OF BYTE := [16#0, 16#04, 16#FF, 16#01, 16#02, 16#03, 16#02, 16#AF, 16#FE];
    cExpectedBytesTest1     : ARRAY[0..31] OF BYTE := [16#FF, 16#01, 16#02, 16#03];
    cExpectedBytesTest2     : ARRAY[0..31] OF BYTE := [16#AF, 16#FE];
END_VAR
TEST(__POUNAME());

ShouldReadBytes(aBuffer:= cRawBytesTest1, aExpectedBytes:= cExpectedBytesTest1, nBufferPosStart:= 1, nExpectedBufferPos:= 6);
ShouldReadBytes(aBuffer:= cRawBytesTest1, aExpectedBytes:= cExpectedBytesTest2, nBufferPosStart:= 6, nExpectedBufferPos:= 9);

TEST_FINISHED_NAMED(__POUNAME());
END_METHOD

END_FUNCTION_BLOCK

// ---- __TESTs/ParsingPrimitivesTests/FB_ReadStringTests.TcPOU
FUNCTION_BLOCK INTERNAL FINAL FB_ReadStringTests EXTENDS FB_TestSuite
VAR_INPUT
END_VAR
VAR_OUTPUT
END_VAR
VAR
END_VAR

ShouldReadStringTheory();

METHOD PRIVATE ShouldReadString
VAR_IN_OUT CONSTANT
    aBuffer         : ARRAY[*] OF BYTE;
    sExpectedString : T_MAXSTRING;
END_VAR
VAR_INPUT CONSTANT
    nBufferPosStart     : UDINT;
    nExpectedBufferPos  : UDINT;
END_VAR
VAR_INST
    fbCtx           : FB_ParseContext;
END_VAR
VAR
    hrActual : HRESULT; 
    // '--- ' to check for null-byte!
    sActual : T_MAXSTRING := '--------------------------------------------------------------------------------------------------------------------------------------------------------------------------------------------------------------------------------------------------------------';
END_VAR

// Arrange
fbCtx.FromBuffer(aBuffer);
fbCtx.refCtx.stState.nBufferPos := nBufferPosStart;

// Act
hrActual := F_ReadString(fbCtx.refCtx, F_ToAnyType(sActual));

// Assert
AssertEquals_DINT(
     Expected:= S_OK,
     Actual:= hrActual,
     Message:= 'Expected S_OK instead of error');
AssertEquals_STRING(
    Expected:= sExpectedString,
    Actual:= sActual,
    Message:= '');
AssertEquals_UDINT(
    Expected:= nExpectedBufferPos,
    Actual:= fbCtx.refCtx.stState.nBufferPos,
    Message:= CONCAT(CONCAT('Expected stState.nBufferPos to equal ', TO_STRING(nExpectedBufferPos)), CONCAT(', for String ', LEFT(sExpectedString, 32))));
END_METHOD

